(* IEC 61131-3 sources: ironplc-benchmarks/compat_out (part 34) *)

(*
version 1.1	15 sep 2007
programmer 	hugo
tested by		tobias

FT_TN7 is delay function, it will delay a signal by a specified time : T and will store 64 values of in before they are put thru to out.
if lower resolution is needed, pls use FT_TN8 or FT_TN16 instead.

*)
(* @END_DECLARATION := '0' *)
(* read system time *)
tx := DWORD_TO_TIME(T_PLC_MS());

trig := FALSE;
IF NOT init THEN
	x[cnt] := in;
	init := TRUE;
	last := tx;
ELSIF tx - last >= T / length THEN
	IF cnt = length - 1 THEN cnt := 0; ELSE cnt := cnt + 1; END_IF;
	Out := X[cnt];
	x[cnt] := in;
	last := tx;
	trig := TRUE;
END_IF;

(* revision history
hm		1. jan 2007		rev 1.0
	original version

hm		16. sep 2007	rev 1.1
	changes time() to T_plc_ms() for compatibility reasons

*)
END_FUNCTION_BLOCK

(* @NESTEDCOMMENTS := 'Yes' *)
(* @PATH := '\/Engineering\/control' *)
(* @OBJECTFLAGS := '0, 8' *)
(* @SYMFILEFLAGS := '2048' *)
FUNCTION_BLOCK FT_TN8
VAR_INPUT
	in : REAL;
	T : TIME;
END_VAR
VAR_OUTPUT
	out : REAL;
	trig: BOOL;
END_VAR
VAR
	length : INT := 8;
	X : ARRAY[0..7] OF REAL;
	cnt : INT;
	last : TIME;
	tx: TIME;
	init: BOOL;
END_VAR

(*
version 1.1	15 Sep 2007
programmer 	hugo
tested by		tobias

FT_TN8 is delay function, it will delay a signal by a specified time : T and will store 8 values of in before they are put thru to out.
if higher resolution is needed, pls use FT_TN16 or FT_TN64 instead.

*)
(* @END_DECLARATION := '0' *)
tx := DWORD_TO_TIME(T_PLC_MS());
trig := FALSE;
IF NOT init THEN
	x[cnt] := in;
	init := TRUE;
	last := tx;
ELSIF tx - last >= T / length THEN
	IF cnt = length - 1 THEN cnt := 0; ELSE cnt := cnt + 1; END_IF;
	Out := X[cnt];
	x[cnt] := in;
	last := tx;
	trig := TRUE;
END_IF;

(* revision history
hm		1. jan 2007		rev 1.0
	original version

hm		16. sep 2007	rev 1.1
	changes time() to T_plc_ms() for compatibility reasons

*)
END_FUNCTION_BLOCK

(* @NESTEDCOMMENTS := 'Yes' *)
(* @PATH := '\/Engineering\/control' *)
(* @OBJECTFLAGS := '0, 8' *)
(* @SYMFILEFLAGS := '2048' *)
FUNCTION_BLOCK HYST
VAR_INPUT
	In : REAL;
	ON : REAL;
	OFF : REAL;
END_VAR
VAR_OUTPUT
	Q : BOOL;
	win : BOOL;
END_VAR

(*
version 1.0	2. jun. 2008
programmer 	hugo
tested BY	oscat

This Hystereses function has two modes:
1. if on > off then Q will be switched high when in > on and switched low when in < off.
2. if on < off then Q will be switched high when in < on and switched low when in > off.
the output win will be high when in is between low and high.

*)
(* @END_DECLARATION := '0' *)
IF ON >= OFF THEN
	IF IN < OFF THEN
		Q := FALSE;
		WIN := FALSE;
	ELSIF  IN > ON THEN
		Q := TRUE;
		WIN := FALSE;
	ELSE
		WIN := TRUE;
	END_IF;
ELSE
	IF IN > OFF THEN
		Q := FALSE;
		WIN := FALSE;
	ELSIF  IN < ON THEN
		Q := TRUE;
		WIN := FALSE;
	ELSE
		WIN := TRUE;
	END_IF;
END_IF;

(* revision history
hm		2.  jun 2008	rev 1.0
	original version

*)
END_FUNCTION_BLOCK

(* @NESTEDCOMMENTS := 'Yes' *)
(* @PATH := '\/Engineering\/control' *)
(* @OBJECTFLAGS := '0, 8' *)
(* @SYMFILEFLAGS := '2048' *)
FUNCTION_BLOCK HYST_1
VAR_INPUT
	In : REAL;
	high : REAL;
	low : REAL;
END_VAR
VAR_OUTPUT
	Q : BOOL;
	win : BOOL;
END_VAR

(*
version 1.1	2. jun. 2008
programmer 	hugo
tested BY	oscat

this hysteresis function switches the output high if the input signal reaches obove high and will switch to low when the input falls back below low value.
a separate output mid is set if the input stays between low and high value.

*)
(* @END_DECLARATION := '0' *)
IF in < low THEN
	Q := FALSE;
	win := FALSE;
ELSIF in > high THEN
	Q := TRUE;
	win := FALSE;
ELSE
	win := TRUE;
END_IF;

(* revision history
hm		4.  aug. 2006	rev 1.0
	original version

hm		2. jun. 2008	rev 1.1
	improved performance
*)
END_FUNCTION_BLOCK

(* @NESTEDCOMMENTS := 'Yes' *)
(* @PATH := '\/Engineering\/control' *)
(* @OBJECTFLAGS := '0, 8' *)
(* @SYMFILEFLAGS := '2048' *)
FUNCTION_BLOCK HYST_2
VAR_INPUT
	IN : REAL;
	VAL : REAL;
	HYS : REAL;
END_VAR
VAR_OUTPUT
	Q : BOOL;
	WIN: BOOL;
END_VAR
VAR
	tmp: REAL;
END_VAR

(*
version 1.2	2. jun. 2008
programmer 	oscat
tested BY	oscat

this hysteresis function switches the output high if the input signal reaches obove val + hys/2 and will switch to low when the input falls back below val - hys/2 value.
a separate output mid is set if the input stays between low and high value.

*)
(* @END_DECLARATION := '0' *)
tmp := val - hys * 0.5;
IF in < tmp THEN
	Q := FALSE;
	win := FALSE;
ELSIF in > tmp + hys THEN
	Q := TRUE;
	win := FALSE;
ELSE
	win := TRUE;
END_IF;

(* revision history
hm		4. aug 2006	rev 1.0
	original version

hm		5. jan 2008	rev 1.1
	improved code for better performance

hm		2. jun. 2008	rev 1.2
	improved performance
*)
END_FUNCTION_BLOCK

(* @NESTEDCOMMENTS := 'Yes' *)
(* @PATH := '\/Engineering\/control' *)
(* @OBJECTFLAGS := '0, 8' *)
(* @SYMFILEFLAGS := '2048' *)
FUNCTION_BLOCK HYST_3
VAR_INPUT
	in : REAL;
	hyst : REAL;
	val1 : REAL;
	val2 : REAL;
END_VAR
VAR_OUTPUT
	Q1 : BOOL;
	Q2 : BOOL;
END_VAR
VAR
	X: REAL;
END_VAR

(*
version 1.2	5 jan 2008
programmer 	oscat
tested BY	oscat

this is a double hysteresis function. Out1 follows a hysteresis function defined by val1and hyst, while out 2 follows val2 and hyst.
if the input signal is between the two hysteresis switches (val1 and val2) then non of the outputs is active.

*)
(* @END_DECLARATION := '0' *)
X := hyst * 0.5;
IF in < val1 - X THEN
	q1 := TRUE;
ELSIF in > val1 + X THEN
	q1 := FALSE;
END_IF;
IF in < val2 - X THEN
	q2 := FALSE;
ELSIF in > val2 + X THEN
	q2 := TRUE;
END_IF;

(* revision history
hm	22. jan 2007	rev 1.0
	original version

hm	27. dec 2007	rev 1.1
	changed code for better performance

hm	5. jan 2008	rev 1.2
	further performance iprovements

*)

END_FUNCTION_BLOCK

(* @NESTEDCOMMENTS := 'Yes' *)
(* @PATH := '\/Engineering\/control' *)
(* @OBJECTFLAGS := '0, 8' *)
(* @SYMFILEFLAGS := '2048' *)
FUNCTION_BLOCK INTEGRATE
VAR_INPUT
	E : BOOL := TRUE;
	X : REAL;
	K : REAL := 1.0;
END_VAR
VAR_IN_OUT
	Y : REAL;
END_VAR
VAR
	X_last : REAL;
	init: BOOL;
	last: DWORD;
	tx: DWORD;
END_VAR

(*
version 1.0	3. nov. 2008
programmer 	hugo
tested by	oscat

integrate is a plain integrator with I/O for out.

*)
(* @END_DECLARATION := '0' *)
(*read system time *)
tx := T_PLC_MS();

IF NOT init THEN
	init := TRUE;
	X_last := X;
ELSIF E THEN
	Y := (X + X_LAST) * 0.5E-3 * DWORD_TO_REAL(tx-last) * K + Y;
	X_last := X;
END_IF;
last := tx;

(*
hm 3. nov. 2008	rev 1.0
original version

*)

END_FUNCTION_BLOCK

(* @NESTEDCOMMENTS := 'Yes' *)
(* @PATH := '\/Engineering\/conversion' *)
(* @OBJECTFLAGS := '0, 8' *)
(* @SYMFILEFLAGS := '2048' *)
FUNCTION_BLOCK ASTRO
VAR_INPUT
	m : REAL;
	AE : REAL;
	PC : REAL;
	LJ : REAL;
END_VAR
VAR_OUTPUT
	Ym : REAL;
	YAE : REAL;
	YPC : REAL;
	YLJ : REAL;
END_VAR

(*
version 1.1	11. mar. 2009
programmer 	hugo
tested by		oscat

this function converts different length units
any unused input can simply be left open.
different inputs connected at the same time will be added up.

*)
(* @END_DECLARATION := '0' *)
YAE :=	AE
		+ m * 6.6845871535E-012
		+ PC * 206265.0
		+ LJ * 63240.0;
Ym := YAE * 149.597870E9;
YPC := YAE * 4.8481322570E-006;
YLJ := YAE * 1.5812776724E-005;

(*
L�nge Meter m SI-Basiseinheit
Astronomische Einheit* AE 1 AE = 149,597 870 � E9 m
Parsec pc 1 pc = 206265 AE = 30,857 � E15 m
Lichtjahr Lj 1 Lj = 9,460 530 � E15 m = 63240 AE = 0,306 59 pc
�ngstr�m � 1 � = E�l0 m
typograph. Punkt p 1 p = 0,376 065 mm � im Druckereigewerbe
inch** in 1 in = 2,54 � E�2 m = 25,4 mm***
foot ft 1 ft = 0,3048 m = 30,48 cm
yard yd 1 yd = 0,9144 m
mile mile 1 mile = 1609,344 m
Internat. Seemeile sm 1 sm = 1852 m
Fathom fm 1 fm = 1,829 m � in der Seeschifffahrt
*)

(* revision history

hm	27. mar. 2007	rev 1.0
	original version

hm	11. mar. 2009	rev 1.1
	improved code

*)

END_FUNCTION_BLOCK

(* @NESTEDCOMMENTS := 'Yes' *)
(* @PATH := '\/Engineering\/conversion' *)
(* @OBJECTFLAGS := '0, 8' *)
(* @SYMFILEFLAGS := '2048' *)
FUNCTION BFT_TO_MS : REAL
VAR_INPUT
	BFT : INT;
END_VAR

(*
version 1.0	12. jun 2008
programmer 	hugo
tested by		oscdat

this function converts wind speed from beaufort to m/s
*)
(* @END_DECLARATION := '0' *)
BFT_TO_MS := EXPT(BFT, 1.5) * 0.836;

(* revision history
hm	12. 6. 2008		rev 1.0
	original version

*)
END_FUNCTION

(* @NESTEDCOMMENTS := 'Yes' *)
(* @PATH := '\/Engineering\/conversion' *)
(* @OBJECTFLAGS := '0, 8' *)
(* @SYMFILEFLAGS := '2048' *)
FUNCTION C_TO_F : REAL
VAR_INPUT
	celsius : REAL;
END_VAR

(*
version 1.1	11. mar. 2009
programmer 	hugo
tested by		tobias

this function converts celsius  to fahrenheit

*)
(* @END_DECLARATION := '0' *)
C_TO_F := celsius * 1.8 + 32.0;

(* revision history

hm	4. aug. 2006	rev 1.0
	original version

hm	11. mar. 2009	rev 1.1
	real constants updated to new systax using dot

*)
END_FUNCTION

(* @NESTEDCOMMENTS := 'Yes' *)
(* @PATH := '\/Engineering\/conversion' *)
(* @OBJECTFLAGS := '0, 8' *)
(* @SYMFILEFLAGS := '2048' *)
FUNCTION C_TO_K : REAL
VAR_INPUT
	Celsius : REAL;
END_VAR

(*
version 1.1	19. aug 2009
programmer 	hugo
tested by		tobias

this function converts celsius to kelvin
*)
(* @END_DECLARATION := '0' *)
C_TO_K := Celsius - phys.T0;

(* revision history

hm	4. aug 2006	rev 1.0
	original version

hm	19. aug 2009	rev 1.1
	fixed calculation error

*)

END_FUNCTION

(* @NESTEDCOMMENTS := 'Yes' *)
(* @PATH := '\/Engineering\/conversion' *)
(* @OBJECTFLAGS := '0, 8' *)
(* @SYMFILEFLAGS := '2048' *)
FUNCTION DEG_TO_DIR : STRING[3]
VAR_INPUT
	DEG : INT;
	N : INT;
	L : INT;
END_VAR
VAR
	ly: INT;
END_VAR

(*
version 1.1	22. oct. 2008
programmer 	hugo
tested by		oscat

this function converts degrees in compass direction.
the function supports output in english (L=0) and german (L=1).

*)
(* @END_DECLARATION := '0' *)
IF L = 0 THEN ly := LANGUAGE.DEFAULT; ELSE ly := MIN(L, LANGUAGE.LMAX); END_IF;
DEG_TO_DIR := LANGUAGE.DIRS[ly, ((SHL(DEG,N-1) + 45) / 90) MOD SHL(INT#2,N)*SHR(INT#8,N)];

(*
DIR := ((SHL(DEG,N-1) + 45) / 90) MOD SHL(INT#2,N);
explanation :
DIR is calculated BY the following formula:
DIR := ((DIR + 45) / 90) MOD 4 if N = 1 digit
North = 0, East = 1 ....
DIR := ((DIR + 22,5) / 45) MOD 8 if N = 2 digit
convert to integer calculation
DIR := ((DIR*2 + 45) / 90) MOD 8
N = 0, NE = 1 ....
ther above formula replaces 2^N with shift for performance
*)

(* revision histroy
hm	11. jun. 2008	rev 1.0
	original release

hm	22. oct. 2008	rev 1.1
	changed size of string variables to 30
*)
END_FUNCTION

(* @NESTEDCOMMENTS := 'Yes' *)
(* @PATH := '\/Engineering\/conversion' *)
(* @OBJECTFLAGS := '0, 8' *)
(* @SYMFILEFLAGS := '2048' *)
FUNCTION DIR_TO_DEG : INT
VAR_INPUT
	DIR : STRING[3];
	L : INT;
END_VAR
VAR
	ly: INT;
	i : INT;
END_VAR

(*
version 1.1	22. oct. 2008
programmer 	hugo
tested by	oscat

this function converts compass directions to degrees
it will recognize up to 3 letter directions in english and german writing.

*)
(* @END_DECLARATION := '0' *)
IF L = 0 THEN ly := LANGUAGE.DEFAULT; ELSE ly := MIN(L, LANGUAGE.LMAX); END_IF;
FOR i := 0 TO 15 DO
	IF language.DIRS[ly, i] = DIR THEN EXIT; END_IF;
END_FOR;
DIR_TO_DEG := SHR(i * 45 + 1, 1);

(* revision histroy
hm	22. oct. 2008	rev 1.1
	original release

*)
END_FUNCTION

(* @NESTEDCOMMENTS := 'Yes' *)
(* @PATH := '\/Engineering\/conversion' *)
(* @OBJECTFLAGS := '0, 8' *)
(* @SYMFILEFLAGS := '2048' *)
FUNCTION_BLOCK ENERGY
VAR_INPUT
	J : REAL;
	C : REAL;
	Wh : REAL;
END_VAR
VAR_OUTPUT
	YJ : REAL;
	YC : REAL;
	YWh : REAL;
END_VAR

(*
version 1.2	16. jan. 2010
programmer 	hugo
tested by		oscat

this function converts different energy units
any unused input can simply be left open.
different inputs connected at the same time will be added up.
*)
(* @END_DECLARATION := '0' *)
YJ := J + Wh * 3600.0 + C * 4.1868;
YC := YJ * 0.238845896627496;
YWh := YJ * 2.7777777778E-004;

(*
Arbeit, Energie, Joule* J 1 J = 1 N � m = 1 W � s = (1/3,6) E�6 kW � h = 1 kg � m2/s2
W�rmemenge Kilowattstunde kW � h 1 kW � h = 3,6 MJ = 860 kcal
Elektronvolt eV 1 eV = 160,218 92 E�21 J
Erg erg 1 erg = 1E�7 J
Kalorie calorie 1 calalorie = 4,1868 J = 1,163 E�3 W � h
Therm therm 1 therm = 105,50 � 106 J
*)

(* revision history

hm	27. mar. 2007	rev 1.0
	original version

hm	11. mar. 2009	rev 1.1
	improved code

hm 16. jan 2010	rev 1.2
	avoid the string cal in comments for codesys import bug

*)
END_FUNCTION_BLOCK

(* @NESTEDCOMMENTS := 'Yes' *)
(* @PATH := '\/Engineering\/conversion' *)
(* @OBJECTFLAGS := '0, 8' *)
(* @SYMFILEFLAGS := '2048' *)
FUNCTION F_TO_C : REAL
VAR_INPUT
	fahrenheit : REAL;
END_VAR

(*
version 1.1	11. mar. 2009
programmer 	hugo
tested BY		tobias

this FUNCTION converts fahrenheit TO celsius

*)
(* @END_DECLARATION := '0' *)
F_TO_C := (fahrenheit - 32.0) * 0.5555555555555;

(* revision history
hm	4. aug 2006	rev 1.0
	original version

hm	11. mar. 2009	rev 1.1
	real constants updated to new systax using dot

*)
END_FUNCTION

(* @NESTEDCOMMENTS := 'Yes' *)
(* @PATH := '\/Engineering\/conversion' *)
(* @OBJECTFLAGS := '0, 8' *)
(* @SYMFILEFLAGS := '2048' *)
FUNCTION F_TO_OM : REAL
VAR_INPUT
	F : REAL;
END_VAR

(*
version 1.1	18. oct. 2008
programmer 	hugo
tested by	oscat

this function converts frequency to Omega F
Omega = 2*PI*F
*)
(* @END_DECLARATION := '0' *)
F_TO_OM := math.PI2 * F;

(* revision history
hm	22. jan. 2007	rev 1.0
	original version

hm	18. oct. 2008	rev 1.1
	unsing math constants

*)
END_FUNCTION

(* @NESTEDCOMMENTS := 'Yes' *)
(* @PATH := '\/Engineering\/conversion' *)
(* @OBJECTFLAGS := '0, 8' *)
(* @SYMFILEFLAGS := '2048' *)
FUNCTION F_TO_PT : TIME
VAR_INPUT
	F : REAL;
END_VAR

(*
version 1.1	11. mar. 2009
programmer 	hugo
tested by		tobias

this function converts frequency to periode time
*)
(* @END_DECLARATION := '0' *)
F_TO_PT := DWORD_TO_TIME(REAL_TO_DWORD(1.0 / F * 1000.0));

(* revision history

hm	4. aug. 2006	rev 1.0
	original version

hm	11. mar. 2009	rev 1.1
	real constants updated to new systax using dot

*)

END_FUNCTION

(* @NESTEDCOMMENTS := 'Yes' *)
(* @PATH := '\/Engineering\/conversion' *)
(* @OBJECTFLAGS := '0, 8' *)
(* @SYMFILEFLAGS := '2048' *)
FUNCTION GEO_TO_DEG : REAL
VAR_INPUT
	D : INT;
	M : INT;
	SEC : REAL;
END_VAR

(*
version 1.0	22. jan. 2009
programmer 	hugo
tested by		oscat

this function converts degrees, minutes seconds to decimal degrees.

*)
(* @END_DECLARATION := '0' *)
GEO_TO_DEG := INT_TO_REAL(D) + INT_TO_REAL(M) * 0.016666666666667 + sec * 0.00027777777777778;

(* revision histroy
hm	22. jan. 2009	rev 1.0
	original release

*)
END_FUNCTION

(* @NESTEDCOMMENTS := 'Yes' *)
(* @PATH := '\/Engineering\/conversion' *)
(* @OBJECTFLAGS := '0, 8' *)
(* @SYMFILEFLAGS := '2048' *)
FUNCTION K_TO_C : REAL
VAR_INPUT
	Kelvin : REAL;
END_VAR

(*
version 1.1	19. aug 2009
programmer 	hugo
tested by		tobias

this function converts kelvin to celsius

*)
(* @END_DECLARATION := '0' *)
K_TO_C := Kelvin + phys.T0;

(* revision history

hm	4. aug 2006	rev 1.0
	original version

hm	19. aug 2009	rev 1.1
	fixed calculation error

*)

END_FUNCTION

(* @NESTEDCOMMENTS := 'Yes' *)
(* @PATH := '\/Engineering\/conversion' *)
(* @OBJECTFLAGS := '0, 8' *)
(* @SYMFILEFLAGS := '2048' *)
FUNCTION KMH_TO_MS : REAL
VAR_INPUT
	kmh : REAL;
END_VAR

(*
version 1.1	6 jan 2007
programmer 	hugo
tested by		tobias

this function converts velocities from Kilometers / hour to Meters / Second

*)
(* @END_DECLARATION := '0' *)
KMH_TO_MS := kmh * 0.2777777777777;

(* revision history
hm	4. feb 2007		rev 1.0
	original version

hm	6. jan 2008		rev 1.1
	improved performance

*)

END_FUNCTION

(* @NESTEDCOMMENTS := 'Yes' *)
(* @PATH := '\/Engineering\/conversion' *)
(* @OBJECTFLAGS := '0, 8' *)
(* @SYMFILEFLAGS := '2048' *)
FUNCTION_BLOCK LENGTH
VAR_INPUT
	m : REAL;
	p : REAL;
	in : REAL;
	ft : REAL;
	yd : REAL;
	mile : REAL;
	sm : REAL;
	fm : REAL;
END_VAR
VAR_OUTPUT
	Ym : REAL;
	Yp : REAL;
	Yin : REAL;
	Yft : REAL;
	Yyd : REAL;
	Ymile : REAL;
	Ysm : REAL;
	Yfm : REAL;
END_VAR

(*
version 1.1	11. mar. 2009
programmer 	hugo
tested by		oscat

this function converts different length units
any unused input can simply be left open.
different inputs connected at the same time will be added up.

*)
(* @END_DECLARATION := '0' *)
Ym :=	m
		+ p * 0.000376065
		+ in * 0.0254
		+ ft * 0.3048
		+ yd * 0.9144
		+ mile * 1609.344
		+ sm * 1852.0
		+ fm * 1.829;
Yp := Ym * 2659.11478068951;
Yin := Ym * 39.37007874016;
Yft := Ym * 3.28083989501;
Yyd := Ym * 1.09361329834;
Ymile := Ym * 0.00062137119;
Ysm := Ym * 0.00053995680;
Yfm := Ym * 0.54674685621;

(*
L�nge Meter m SI-Basiseinheit
Astronomische Einheit* AE 1 AE = 149,597 870 � E9 m
Parsec pc 1 pc = 206265 AE = 30,857 � E15 m
Lichtjahr Lj 1 Lj = 9,460 530 � E15 m = 63240 AE = 0,306 59 pc
�ngstr�m � 1 � = E�l0 m
typograph. Punkt p 1 p = 0,376 065 mm � im Druckereigewerbe
inch** in 1 in = 2,54 � E�2 m = 25,4 mm***
foot ft 1 ft = 0,3048 m = 30,48 cm
yard yd 1 yd = 0,9144 m
mile mile 1 mile = 1609,344 m
Internat. Seemeile sm 1 sm = 1852 m
Fathom fm 1 fm = 1,829 m � in der Seeschifffahrt
*)

(* revision history

hm	27. mar. 2007	rev 1.0
	original version

hm	11. mar. 2009	rev 1.1
	improved code

*)

END_FUNCTION_BLOCK

(* @NESTEDCOMMENTS := 'Yes' *)
(* @PATH := '\/Engineering\/conversion' *)
(* @OBJECTFLAGS := '0, 8' *)
(* @SYMFILEFLAGS := '2048' *)
FUNCTION MS_TO_BFT : INT
VAR_INPUT
	MS : REAL;
END_VAR

(*
version 1.0	12. jun 2008
programmer 	hugo
tested by	oscdat

this function converts wind speed from M/s to beaufort
*)
(* @END_DECLARATION := '0' *)
MS_TO_BFT := REAL_TO_INT(EXPT(MS * 1.196172, 0.666667));

(* revision history
hm	12. 6. 2008		rev 1.0
	original version

*)
END_FUNCTION

(* @NESTEDCOMMENTS := 'Yes' *)
(* @PATH := '\/Engineering\/conversion' *)
(* @OBJECTFLAGS := '0, 8' *)
(* @SYMFILEFLAGS := '2048' *)
FUNCTION MS_TO_KMH : REAL
VAR_INPUT
	ms : REAL;
END_VAR

(*
version 1.0	4 Feb 2007
programmer 	hugo
tested by		tobias

this function converts velocities from Meters / Second to Kilometers / hour.

*)
(* @END_DECLARATION := '0' *)
MS_TO_KMH := ms * 3.6;

END_FUNCTION

(* @NESTEDCOMMENTS := 'Yes' *)
(* @PATH := '\/Engineering\/conversion' *)
(* @OBJECTFLAGS := '0, 8' *)
(* @SYMFILEFLAGS := '2048' *)
FUNCTION OM_TO_F : REAL
VAR_INPUT
	OM : REAL;
END_VAR

(*
version 1.1	18. oct. 2008
programmer 	hugo
tested by		tobias

this function converts Omega F to frequency
F = OM / (2*PI)
*)
(* @END_DECLARATION := '0' *)
OM_TO_F := OM / math.PI2;

(* revision history
hm	22. jan. 2007	rev 1.0
	original version

hm	18. oct. 2008	rev 1.1
	using math constants

*)
END_FUNCTION

(* @NESTEDCOMMENTS := 'Yes' *)
(* @PATH := '\/Engineering\/conversion' *)
(* @OBJECTFLAGS := '0, 8' *)
(* @SYMFILEFLAGS := '2048' *)
FUNCTION_BLOCK PRESSURE
VAR_INPUT
	mws : REAL;
	torr : REAL;
	att : REAL;
	atm : REAL;
	pa : REAL;
	bar : REAL;
END_VAR
VAR_OUTPUT
	Ymws : REAL;
	Ytorr : REAL;
	Yatt : REAL;
	Yatm : REAL;
	Ypa : REAL;
	Ybar : REAL;
END_VAR

(*
version 1.1	11. mar. 2009
programmer 	hugo
tested by		oscat

this function converts different pressure units
any unused input can simply be left open.
different inputs connected at the same time will be added up.
*)
(* @END_DECLARATION := '0' *)
Ybar := bar +
		pa * 1.0E-5 +
		0.980665 * att +
		1.01325 * atm +
		0.001333224 * torr +
		0.0980665 * mws;
Ymws := ybar * 10.1971621297793;
Ytorr := ybar * 750.0615050434140;
Yatt := ybar * 1.0197162129779;
yatm := ybar * 0.9869232667160;
Ypa := ybar * 100000.0;

(*
Druck, Pascal Pa 1 Pa = 1 N/m2 = 1 kg/(s2 �E m) . 0,75 �E 10.2 mmHg
mechanische 1 MPa = 1 N/mm2 . fur Festigkeitsangaben
Spannung Bar bar 1 bar = 105 Pa = 103 mbar = 105 kg/(s2 �E m)
Millimeter- mmHg 1 mmHg = 133,322 Pa = 1,333 22 mbar
Quecksilbersaule . nur in Heilkunde zulassig
physik. Atmosphare atm 1 atm = 1,013 25 bar
techn. Atmosphare at 1 at = 1 kp/cm2 = 0,980665 bar
Torr Torr 1 Torr = (101325/760) Pa = 1,333224 mbar
Meter-Wassersaule mWS 1 mWS = 9806,65 Pa = 98,0665 mbar
psi lbf/in2 1 lbf/in2 = 68,947 57 mbar = 6894,757 Pa

*)

(* revision history

hm	27. mar. 2007	rev 1.0
	original version

hm	11. mar. 2009	rev 1.1
	improved code

*)
END_FUNCTION_BLOCK

(* @NESTEDCOMMENTS := 'Yes' *)
(* @PATH := '\/Engineering\/conversion' *)
(* @OBJECTFLAGS := '0, 8' *)
(* @SYMFILEFLAGS := '2048' *)
FUNCTION PT_TO_F : REAL
VAR_INPUT
	PT : TIME;
END_VAR

(*
version 1.1	11. mar. 2009
programmer 	hugo
tested by		tobias

this function converts periode time to frequency
*)
(* @END_DECLARATION := '0' *)
PT_TO_F := 1000.0 / DWORD_TO_REAL(TIME_TO_DWORD(PT));

(*	revision history
hm	4. aug. 2006	rev 1.0
	original version

hm	11. mar. 2009	rev 1.1
	real constants updated to new systax using dot

*)

END_FUNCTION

(* @NESTEDCOMMENTS := 'Yes' *)
(* @PATH := '\/Engineering\/conversion' *)
(* @OBJECTFLAGS := '0, 8' *)
(* @SYMFILEFLAGS := '2048' *)
FUNCTION_BLOCK SPEED
VAR_INPUT
	ms : REAL;
	kmh : REAL;
	kn : REAL;
	mh : REAL;
END_VAR
VAR_OUTPUT
	Yms : REAL;
	Ykmh : REAL;
	Ykn : REAL;
	Ymh : REAL;
END_VAR

(*
version 1.1	11. mar. 2009
programmer 	hugo
tested by		oscat

this function converts different speed units
any unused input can simply be left open.
different inputs connected at the same time will be added up.

*)
(* @END_DECLARATION := '0' *)
Yms := ms +
		kmh * 0.27777777777778 +
		kn * 0.5144444 +
		mh * 0.44704;
Ykmh := Yms * 3.6;
Ykn := Yms * 1.94384466037535;
Ymh := Yms * 2.23693629205440;

(*
Geschwindigkeit Meter durch Sekunde m/s 1 m/s = 3,6 km/h
km durch (pro) Stunde, nicht �Stundenkilometer� verwenden
Knoten kn 1 kn = 1 sm/h = 0,5144 m/s

*)

(* revision history
hm	27. mar. 2009	rev 1.0
	original version

hm	11. mar. 2009	rev 1.1
	improved code

*)
END_FUNCTION_BLOCK

(* @NESTEDCOMMENTS := 'Yes' *)
(* @PATH := '\/Engineering\/conversion' *)
(* @OBJECTFLAGS := '0, 8' *)
(* @SYMFILEFLAGS := '2048' *)
FUNCTION_BLOCK TEMPERATURE
VAR_INPUT
	K : REAL;
	C : REAL := -273.15;
	F : REAL := -459.67;
	Re : REAL := -218.52;
	Ra : REAL;
END_VAR
VAR_OUTPUT
	YK : REAL;
	YC : REAL;
	YF : REAL;
	YRe : REAL;
	YRa : REAL;
END_VAR

(*
version 1.0	21 feb 2008
programmer 	hugo
tested by	oscat

this function converts different temperature units
any unused input can simply be left open.
different inputs connected at the same time will be added up.

*)
(* @END_DECLARATION := '0' *)
YK := K + (C + 273.15) + (F + 459.67) * 0.555555555555 + (Re * 1.25 + 273.15) + (Ra * 0.555555555555);
YC := YK -273.15;
YF := YK * 1.8 - 459.67;
YRe := (YK - 273.15) * 0.8;
YRa := YK * 1.8;

(* revision history
hm	21. feb. 2008	rev 1.0
	original version

*)
END_FUNCTION_BLOCK

(* @NESTEDCOMMENTS := 'Yes' *)
(* @PATH := '\/Engineering\/measurements' *)
(* @OBJECTFLAGS := '0, 8' *)
(* @SYMFILEFLAGS := '2048' *)
FUNCTION_BLOCK ALARM_2
VAR_INPUT
	X : REAL;
	LO_1 : REAL;
	HI_1 : REAL;
	LO_2 : REAL;
	HI_2 : REAL;
	HYS : REAL;
END_VAR
VAR_OUTPUT
	Q1_LO : BOOL;
	Q1_HI : BOOL;
	Q2_LO : BOOL;
	Q2_HI : BOOL;
END_VAR
VAR
	tmp: REAL;
END_VAR

(*
	version 1.1	11. mar. 2009
	programmer 	hugo
	tested BY		tobias

ALARM_2 will check two pairs of limits and signal when the input is above or below a set limit.
with the input HYS a hysteresis can be defined for all limits.

*)
(* @END_DECLARATION := '0' *)
tmp := X - Hys * 0.5;
IF tmp > LO_1 THEN Q1_LO := FALSE; END_IF;
IF tmp > LO_2 THEN Q2_LO := FALSE; END_IF;
IF tmp > HI_1 THEN Q1_HI := TRUE; END_IF;
IF tmp > HI_2 THEN Q2_HI := TRUE; END_IF;
tmp := tmp + hys;
IF tmp < LO_1 THEN Q1_LO := TRUE; END_IF;
IF tmp < LO_2 THEN Q2_LO := TRUE; END_IF;
IF tmp < HI_1 THEN Q1_HI := FALSE; END_IF;
IF tmp < HI_2 THEN Q2_HI := FALSE; END_IF;

(* revision history
hm	19. may. 2008		rev 1.0
	original version

hm	11. mar. 2009	rev 1.1
	improved code
*)

END_FUNCTION_BLOCK

(* @NESTEDCOMMENTS := 'Yes' *)
(* @PATH := '\/Engineering\/measurements' *)
(* @OBJECTFLAGS := '0, 8' *)
(* @SYMFILEFLAGS := '2048' *)
FUNCTION_BLOCK BAR_GRAPH
VAR_INPUT
	X : REAL;
	rst : BOOL;
END_VAR
VAR_INPUT (* CONSTANT *)
	trigger_Low : REAL;
	trigger_High : REAL;
	Alarm_low : BOOL;
	Alarm_high : BOOL;
	log_scale : BOOL;
END_VAR
VAR_OUTPUT
	LOW, Q1, Q2, Q3, Q4, Q5, Q6, HIGH : BOOL;
	Alarm : BOOL;
	Status : BYTE;
END_VAR
VAR
	init : BOOL;
	T1, T2, T3, T4, T5 : REAL;
END_VAR
VAR_TEMP
	temp : REAL;
END_VAR

(*
	version 1.2	6 jan 2008
	programmer 	hugo
	tested BY	hans

bar graph is a muti window comparator which displays an analog input signal on 8 digital outputs.
only one output is active a any given time depending on the value of the input signal.
the output can be of linear or logarithmic scale.

*)
(* @END_DECLARATION := '0' *)
IF NOT init THEN
	init := TRUE;
	IF log_scale THEN
		temp := EXP(LN(Trigger_high / Trigger_low) * 0.166666666666666666666);
		T1 := trigger_low * temp;
		T2 := T1 * temp;
		T3 := T2 * temp;
		T4 := T3 * temp;
		T5 := T4 * temp;
	ELSE
		temp := (trigger_high - trigger_low) * 0.142857142;
		T1 := trigger_low + temp;
		T2 := T1 + temp;
		T3 := T2 + temp;
		T4 := T3 + temp;
		T5 := T4 + temp;
	END_IF;
END_IF;

(* clear outputs before checking *)
Q1 := FALSE;
Q2 := FALSE;
Q3 := FALSE;
Q4 := FALSE;
Q5 := FALSE;
Q6 := FALSE;
status := 110;

(* low, high and alarm can only be cleared with rst depending on alarm_low and alarm_high *)
IF NOT alarm_low THEN low := FALSE; END_IF;
IF NOT alarm_high THEN high := FALSE; END_IF;
IF rst THEN
	alarm := FALSE;
	low := FALSE;
	high := FALSE;
END_IF;

(* check and set outputs *)
IF X < trigger_low THEN
	Low := TRUE;
	status := 111;
	IF alarm_low THEN
		alarm := TRUE;
		status := 1;
	END_IF;
ELSIF X < T1 THEN
	Q1 := TRUE;
ELSIF x < t2 THEN
	Q2 := TRUE;
ELSIF x < t3 THEN
	Q3 := TRUE;
ELSIF x < T4 THEN
	Q4 := TRUE;
ELSIF x < T5 THEN
	q5 := TRUE;
ELSIF x < trigger_high THEN
	q6 := TRUE;
ELSE
	high := TRUE;
	status := 112;
	IF alarm_high THEN
		alarm := TRUE;
		status := 2;
	END_IF;
END_IF;

(* revision history
hm	22. feb 2007	rev 1.0
	original version

hm	2. dec 2007		rev 1.1
	chaged code for better performance

hm	6. jan 2008		rev 1.2
	further performance improvement

*)
END_FUNCTION_BLOCK

(* @NESTEDCOMMENTS := 'Yes' *)
(* @PATH := '\/Engineering\/measurements' *)
(* @OBJECTFLAGS := '0, 8' *)
(* @SYMFILEFLAGS := '2048' *)
FUNCTION_BLOCK CALIBRATE
VAR_INPUT
	X : REAL;
	CO : BOOL;
	CS : BOOL;
END_VAR
VAR_INPUT (* CONSTANT *)
	Y_Offset : REAL;
	Y_Scale : REAL;
END_VAR
VAR_OUTPUT
	Y : REAL;
END_VAR
VAR RETAIN
	offset : REAL;
	Scale : REAL := 1.0;
END_VAR

(*
	version 1.3	11. mar. 2009
	programmer 	hugo
	tested BY		hans

Calibrate allows for offset and scale calibration of an analog input.
offset is calibrated to a stored reference Y_offset while CO is true.
after the offset is calibrated, scale can be calibrated to a reference value Y_scale while CS is true.
*)
(* @END_DECLARATION := '0' *)
(* check for calibration *)
IF CO THEN
	OFFSET := Y_Offset - X;
ELSIF CS THEN
	SCALE := Y_scale / (X + OFFSET);
END_IF;
(* calculate output *)
Y := (X + OFFSET) * SCALE;

(* revision history
hm 22.2.2007		rev 1.2
	changed VAR RETAIN PERSISTENT to VAR RETAIN for better compatibility
	wago lon contollers do not support persisitent

hm	11. mar. 2009	rev 1.3
	changed real constants to use dot syntax

*)
END_FUNCTION_BLOCK

(* @NESTEDCOMMENTS := 'Yes' *)
(* @PATH := '\/Engineering\/measurements' *)
(* @OBJECTFLAGS := '0, 8' *)
(* @SYMFILEFLAGS := '2048' *)
FUNCTION_BLOCK CYCLE_TIME
VAR_INPUT
	RST : BOOL;
END_VAR
VAR_OUTPUT
	ct_min : TIME;
	ct_max : TIME;
	ct_last : TIME;
	systime : TIME;
	sysdays : INT;
	cycles : DWORD;
END_VAR
VAR
	last_cycle : TIME;
	tx: TIME;
	init: BOOL;
END_VAR

(*
	version 1.2	16 sep 2007
	programmer 	hugo
	tested BY		hans

this function block measures the cycle time and displays the last, min and max cycle time of the current task.
the resolution is 1ms.
the cycles output is a dword counter which counts the cycles.
a rst pulse on the input will reset all data.

*)
(* @END_DECLARATION := '0' *)
tx := DWORD_TO_TIME(T_PLC_MS()) - last_cycle;
IF rst THEN
	ct_min := t#10h;
	ct_max := t#0ms;
	cycles := 0;
ELSIF last_cycle > t#0s THEN
	IF tx < ct_min THEN ct_min := tx;
	ELSIF tx > ct_max THEN ct_max := tx;
	END_IF;
	ct_last := tx;
ELSIF ct_min = t#0s THEN
	ct_min := t#0s - t#1ms;
END_IF;
IF init THEN
	systime := systime + tx;
		IF systime >= t#1d THEN
			systime := systime - t#1d;
			sysdays := sysdays + 1;
		END_IF;
END_IF;
init := TRUE;
last_cycle := last_cycle + tx;
cycles := cycles + 1;

(*	revision history
hm 12.12.2006		rev 1.1
	added cycles output, a dword cycle counter.
hm 10.3.2007			rev 1.2
	changed initialization of ct_min to t#10h for compatibility with siemens s7

hm	16.9.2007		rev 1.2
	changed Time() in T_PLC_MS() for compatibility resons

*)
END_FUNCTION_BLOCK

(* @NESTEDCOMMENTS := 'Yes' *)
(* @PATH := '\/Engineering\/measurements' *)
(* @OBJECTFLAGS := '0, 8' *)
(* @SYMFILEFLAGS := '2048' *)
FUNCTION_BLOCK DT_SIMU
VAR_INPUT
	START : DT;
	SPEED : REAL := 1.0;
END_VAR
VAR_OUTPUT
	DTS : DT;
END_VAR
VAR
	tc : DWORD;
	init: BOOL;
	last: DWORD;
	tx: DWORD;
	td: DWORD;
END_VAR

(*
version 1.2	8. mar. 2009
programmer 	hugo
tested by		oscat

DT_SIMU simulates a real time clock and can be adjusted to different speeds
it can also be used in simulation to simulate a real time clock.
the peed of the clock can be increased or decreased to debug timers.
with the input start a start date-time can be specified.

*)
(* @END_DECLARATION := '0' *)
(* read system timer *)
tx := T_PLC_MS();
tc := REAL_TO_DWORD(DWORD_TO_REAL(tx - last) * speed);

IF NOT init THEN
	init := TRUE;
	DTS := Start;
	tc := 0;
	last := tx;
ELSIF SPEED = 0.0 THEN
	DTS := DWORD_TO_DT(DT_TO_DWORD(DTS) + 1);
ELSIF tc >= 1000 THEN
	td := (tc / 1000) * 1000;
	DTS := DTS + DWORD_TO_TIME(td);
	last := last + REAL_TO_DWORD(DWORD_TO_REAL(td) / speed);
END_IF;

(* revision history
hm	11. sep. 2008	rev 1.0
	original version

hm	16. nov	2008	rev 1.1
	added type conversions for compatibility reasons

hm	8.	mar. 2009	rev 1.2
	added increment by cycle mode

*)

END_FUNCTION_BLOCK

(* @NESTEDCOMMENTS := 'Yes' *)
(* @PATH := '\/Engineering\/measurements' *)
(* @OBJECTFLAGS := '0, 8' *)
(* @SYMFILEFLAGS := '2048' *)
FUNCTION_BLOCK FLOW_METER
VAR_INPUT
	VX : REAL;
	E : BOOL;
	RST : BOOL;
END_VAR
VAR_INPUT (* CONSTANT *)
	PULSE_MODE : BOOL;
	UPDATE_TIME : TIME := t#1s;
END_VAR
VAR_OUTPUT
	F : REAL;
END_VAR
VAR_IN_OUT
	X : REAL;
	Y : UDINT;
END_VAR
VAR
	tx, tl : TIME;
	int1 : INTEGRATE;
	init: BOOL;
	e_last : BOOL;
	tmp: INT;
	x_last : REAL;
	y_last : UDINT;
END_VAR

(*
version 1.0	23. jan. 2011
programmer 	hugo
tested by	oscat

Flow meter measures flow according to gated time or pulses.

*)

(* @END_DECLARATION := '0' *)
IF NOT init THEN	(* init on power up *)
	init := TRUE;
	tl := tx;
	x_last := X;
	y_last := Y;
	int1.K := 2.7777777777777777E-4;
END_IF;

(* run integrator *)
int1(E := NOT (RST OR PULSE_MODE) AND E, X := VX, Y := X);	(* gated operation *)

IF RST THEN		(* reset *)
	X := 0.0;
	Y := 0;
	tl := tx;
	x_last := 0.0;
	y_last := 0;
ELSIF E AND PULSE_MODE THEN	(* check for pulse mode *)
	IF NOT e_last THEN X := X + VX; END_IF;
END_IF;
e_last := E;

(* reduce X to be less than 1 and increase Y respectively *)
IF X > 1.0 THEN
	tmp := FLOOR(X);
	Y := Y + INT_TO_UDINT(tmp);
	X := X - INT_TO_REAL(tmp);
END_IF;

(* calculate the current flow *)
tx := DWORD_TO_TIME(T_PLC_MS());
IF tx - tl >= UPDATE_TIME AND UPDATE_TIME > t#0s THEN
	F := (UDINT_TO_REAL(Y - y_last) + X - x_last) / TIME_TO_REAL(tx - tl) * 3.6E6;
	y_last := Y;
	x_last := X;
	tl := tx;
END_IF;

(* revision history
hm	23. jan. 2011	rev 1.0
	original version

*)

END_FUNCTION_BLOCK

(* @NESTEDCOMMENTS := 'Yes' *)
(* @PATH := '\/Engineering\/measurements' *)
(* @OBJECTFLAGS := '0, 8' *)
(* @SYMFILEFLAGS := '2048' *)
FUNCTION_BLOCK M_D
VAR_INPUT
	start : BOOL;
	stop : BOOL;
	tmax : TIME := t#10d;
	rst: BOOL;
END_VAR
VAR_OUTPUT
	PT : TIME;
	ET : TIME;
	run : BOOL;
END_VAR
VAR
	edge : BOOL;
	T0 : TIME;
	tx: TIME;
	startup: BOOL;
END_VAR

(*
	version 1.2	27. feb. 2009
	programmer 	hugo
	tested BY	oscat

m_d measures the time between a rising edge on start to a rising edge on stop and returs the last measured value on the output PT.
a second output ET is starting from 0 at the rising edge of start and is counting up until the rising edge of stop occurs.
the asynchronous input rst can reset the outputs at any time.
tmax defines a timeout wich is the maximum measurable time between start and stop, if this time is exceeded the outputs will stay at 0.
*)
(* @END_DECLARATION := '0' *)
(* check for rst input *)
IF rst OR et >= tmax THEN
	pt := t#0ms;
	et := t#0ms;
	startup := FALSE;
	run := FALSE;
END_IF;

(* avoid timers to start when input is true at startup *)
IF NOT startup THEN
	edge := start;
	startup := TRUE;
END_IF;

(* read system timer *)
tx := DWORD_TO_TIME(T_PLC_MS());

(* detect rising edge on start *)
IF start AND NOT edge AND NOT stop THEN
	t0 := tx;
	run := TRUE;
	pt := t#0s;
ELSIF stop AND run THEN
	pt := et;
	run := FALSE;
END_IF;
edge := start;
IF run THEN et := tx - t0; END_IF;

(* revision history
hm		2.5.2007	rev 1.0
	original version

hm		16.9.2007	rev 1.1
	changes time() to T_plc_ms() for compatibility reasons

hm	27. feb 2009	rev 1.2
	deleted unnecessary init with 0
*)

END_FUNCTION_BLOCK

(* @NESTEDCOMMENTS := 'Yes' *)
(* @PATH := '\/Engineering\/measurements' *)
(* @OBJECTFLAGS := '0, 8' *)
(* @SYMFILEFLAGS := '2048' *)
FUNCTION_BLOCK M_T
VAR_INPUT
	IN : BOOL;
	TMAX : TIME := t#10d;
	RST : BOOL;
END_VAR
VAR_OUTPUT
	PT : TIME;
	ET: TIME;
END_VAR
VAR
	edge : BOOL;
	start : TIME;
	tx: TIME;
END_VAR

(*
version 1.4	10. mar. 2009
programmer 	hugo
tested BY		oscat

m_t measures the with of a high pulse and returs the last measured pulse width on output PT.
a second output ET is starting from 0 at the rising edge and counting up until the falling edge occurs and resetts et to 0.
the asynchrtonous input rst can reset the outputs at any time.
tmax defines a maximum measurable time, if this value is exceeded the outputs will be reset to 0.

*)
(* @END_DECLARATION := '0' *)
(* read system time *)
tx := DWORD_TO_TIME(T_PLC_MS());

IF RST OR ET >= TMAX THEN
	PT :=  t#0s;
	ET := t#0s;
ELSIF IN THEN
	IF NOT edge THEN start := tx; END_IF;
	ET := tx - start;
ELSE
	PT := ET;
END_IF;
edge := IN;

(* revision history
hm	4. aug. 2006	rev 1.0
	original version

hm	2. may. 2007	rev 1.1
	added init variable to avoid unreasonable measurement if falling edge occurs first.
	added et (elapsed time) output to count from 0 at rising edge until a falling edge resets et to 0.
	added reset input.

hm	16. sep. 2007	rev 1.2
	changes time() to T_plc_ms() for compatibility reasons

hm	17. dec. 2008	rev 1.3
	code optimized

hm	10. mar. 2009	rev 1.4
	removed nested comments
	removed double assignments

*)
END_FUNCTION_BLOCK

(* @NESTEDCOMMENTS := 'Yes' *)
(* @PATH := '\/Engineering\/measurements' *)
(* @OBJECTFLAGS := '0, 8' *)
(* @SYMFILEFLAGS := '2048' *)
FUNCTION_BLOCK M_TX
VAR_INPUT
	in: BOOL;
	tmax : TIME := t#10d;
	rst : BOOL;
END_VAR
VAR_OUTPUT
	TH : TIME;
	TL : TIME;
	DC : REAL;
	F: REAL;
	ET : TIME;
END_VAR
VAR
	edge : BOOL;
	start: TIME;
	stop:TIME;
	tx: TIME;
	rise : BOOL;
	fall : BOOL;
	startup: BOOL;
END_VAR

(*
	version 1.4	11. mar. 2009
	programmer 	oscat
	tested BY		oscat

this measures the timing of a signal
TH is the high pulse width
TL is the low pulse width
DC is the duty cycle
F is the frequency
ET will start at 0 with a rising edge and count up till the next rising edge starts from 0 again.
the acuracy depends on the cycle time of the sps and is limited to 1ms resolution.
an asynchronous reset can reset all outputs to 0 at any time.
the input tmax can configure a timeout for ET where the function block will outomatically reset itself.
tmx is predefined to 10 days.
*)
(* @END_DECLARATION := '0' *)
(* check FOR rst input *)
IF rst OR (et >= tmax) THEN
	rise := FALSE;
	fall := FALSE;
	startup := FALSE;
	th := t#0ms;
	tl := t#0ms;
	DC := 0.0;
	F := 0.0;
	ET := t#0s;
END_IF;

(* avoid timers to start when input is true at startup *)
IF NOT startup THEN
	edge := in;
	startup := TRUE;
END_IF;

(* read system timer *)
tx := DWORD_TO_TIME(T_PLC_MS());

(* edge trigger rising and falling edge *)
IF in XOR edge THEN
	edge := in;
	(* rising edge starts measurement *)
	IF in THEN
		start := Tx;
		rise := TRUE;
		IF fall THEN tl := start - stop; END_IF;
		IF th > t#0ms AND tl > t#0ms THEN
			dc := TIME_TO_REAL(th) / TIME_TO_REAL(th+tl);
			f := 1000.0 / TIME_TO_REAL(th + tl);
		END_IF;
	(* falling edge starts second cycle measurement *)
	ELSE
		stop := Tx;
		fall := TRUE;
		IF rise THEN th := stop - start; END_IF;
		IF th > t#0ms AND tl > t#0ms THEN
			dc := TIME_TO_REAL(th) /  TIME_TO_REAL(th+tl);
			f := 1000.0 / TIME_TO_REAL(th + tl);
		END_IF;
	END_IF;
END_IF;
IF rise THEN et := tx - start; END_IF;

(* revision history
hm	4. aug. 2006	rev 1.0
	original version

hm	2. mai. 2007	rev 1.1
	made sure that no undefined values would be measured at startup conditions
	added output et
	added rst input
	added tmax input

hm	16. sep. 2007	rev 1.2
	changes time() to T_plc_ms() for compatibility reasons

hm	27. feb. 2009	rev 1.3
	deleted unnecessary init with 0

hm	11. mar. 2009	rev 1.4
	changed real constants to use dot syntax

*)
END_FUNCTION_BLOCK

(* @NESTEDCOMMENTS := 'Yes' *)
(* @PATH := '\/Engineering\/measurements' *)
(* @OBJECTFLAGS := '0, 8' *)
(* @SYMFILEFLAGS := '2048' *)
FUNCTION_BLOCK METER
VAR_INPUT
	M1, M2 : REAL;
	I1, I2 : BOOL;
	D : REAL := 1.0;
	RST : BOOL;
END_VAR
VAR_IN_OUT
	MX : REAL;
END_VAR
VAR
	MR : REAL2;
	MX1, MX2 : REAL; (* current consumption value on M1 and M2 *)
	tx: DWORD;
	last: DWORD;
	tc: REAL;
	init: BOOL;
END_VAR

(*
	version 1.4	8. mar. 2009
	programmer 	oscat
	tested BY	oscat

METER measures usage of power or similar values the output MX is the sum of the inputs over time.
MX := sum over time of (I1 * P1 + I2 * P2)/D.
a simple example is the consumption counter for a 2 stage oil burner where stage 1 is 10KW and stage 2 is 20KW.
I1 and I2 decide which value is accounted for, I1 = True only counts P1, I2 is True counts P2
and I1 and I2 is true counts P1 and P2.
the meter can be used for all kind of consumption meters. P1 and P2 can change on the fly.

*)
(* @END_DECLARATION := '0' *)
(* measure the last cycle time and make sure we onle execute once every millisecond *)
tx := T_PLC_MS();
IF NOT init THEN
	init := TRUE;
	last := tx;
	mr.RX := mx;
	mr.R1 := 0.0;
ELSIF tx = last THEN
	RETURN;
ELSE
	tc := DWORD_TO_REAL(tx - last) * 0.001;
END_IF;
last := tx;

(* reset *)
IF rst THEN
	mr.R1 := 0.0;
	mr.RX := 0.0;
ELSE
	(* current consumption measurement *)
	IF I1 THEN MX1 := M1; ELSE MX1 := 0.0; END_IF;
	IF I2 THEN MX2 := M2; ELSE MX2 := 0.0; END_IF;
	(* add up the current values in a double real *)
	MR := R2_ADD(MR,(SEL(I1,0.0,mx1) + SEL(I2, 0.0, mx2)) / D * TC);
	(* set the current output value *)
	MX := mr.RX;
END_IF;

(* revision history

hm	16. sep.2007		rev 1.0
	original version

hm	7. feb 2008		rev 1.1
	use new version of ft_int to avoid a counting stop at high values
	deleted unnecessary limits

hm	24. mar. 2008	rev 1.2
	use data_type real2 to extend accuracy to 15 digits total
	do not use ft_int which adds unnecessary overhead

hm	8. feb. 2009	rev 1.3
	changed mx to be I/O
	make sure calculation works for cycle times < 1 ms

hm	8. mar. 2009	rev 1.4
	last was not updated
	code improvements

*)

END_FUNCTION_BLOCK

(* @NESTEDCOMMENTS := 'Yes' *)
(* @PATH := '\/Engineering\/measurements' *)
(* @OBJECTFLAGS := '0, 8' *)
(* @SYMFILEFLAGS := '2048' *)
FUNCTION_BLOCK METER_STAT
VAR_INPUT
	IN : REAL;
	DI : DATE;
	RST : BOOL;
END_VAR
VAR_IN_OUT
	Last_Day : REAL;
	Current_Day : REAL;
	Last_Week : REAL;
	Current_Week : REAL;
	Last_Month : REAL;
	Current_Month : REAL;
	Last_Year : REAL;
	Current_Year : REAL;
END_VAR
VAR RETAIN
	Year_Start : REAL;
	Month_Start : REAL;
	Week_Start : REAL;
	Day_Start : REAL;
	last_run: DATE;
END_VAR

(*
	version 1.3	18. jul. 2009
	programmer 	oscat
	tested BY		oscat

METER_STAT runs statistics of a metered value, it calculates the current week, day, month and year consumption and stores the corresponding last day, week, month and year value.

*)
(* @END_DECLARATION := '0' *)
IF rst THEN
	Last_Day := 0.0;
	Current_Day := 0.0;
	Day_start := IN;
	Last_week := 0.0;
	Current_week := 0.0;
	Week_start := in;
	Last_month := 0.0;
	Current_month := 0.0;
	month_start := in;
	last_year := 0.0;
	current_year := 0.0;
	year_start := in;
ELSE
	Current_Day := IN - Day_Start;
	Current_Week := In - Week_Start;
	Current_Month := IN - Month_Start;
	Current_Year := IN - Year_Start;
END_IF;

IF YEAR_OF_DATE(DI) > YEAR_OF_DATE(last_run) THEN
	(* a new year has started *)
	last_year := current_year;
	current_year := 0.0;
	year_start := in;
	last_month := current_month;
	current_month := 0.0;
	month_start := in;
	last_day := current_day;
	current_day := 0.0;
	day_start := in;
ELSIF MONTH_OF_DATE(DI) > MONTH_OF_DATE(last_run) THEN
	(* a new month has started, january is alrerady done by year change *)
	last_month := current_month;
	current_month := 0.0;
	month_start := in;
	last_day := current_day;
	current_day := 0.0;
	day_start := in;
ELSIF DAY_OF_YEAR(di) > DAY_OF_YEAR(last_run) THEN
	(* day has chaged, first day of year and first day of month has already been taken care of *)
	last_day := current_day;
	current_day := 0.0;
	day_start := in;
END_IF;
IF DAY_OF_WEEK(DI) < DAY_OF_WEEK(last_run) THEN
	(* a new week has started *)
	last_week := current_week;
	current_week := 0.0;
	week_start := in;
END_IF;
last_run := di;

(* revision history
hm	16. sep. 2007	rev 1.0
	original version

hm	7. oct. 2008	rev 1.1
	changed function year_to_year_of_date
	changed function month to month_of_date
	changed function weekday to day_of_week

hm	11. mar. 2009	rev 1.2
	changed real constants to use dot syntax

hm	18. jul. 2009	rev 1.3
	changes all outputs to be I/O
*)

END_FUNCTION_BLOCK

(* @NESTEDCOMMENTS := 'Yes' *)
(* @PATH := '\/Engineering\/measurements' *)
(* @OBJECTFLAGS := '0, 8' *)
(* @SYMFILEFLAGS := '2048' *)
FUNCTION_BLOCK ONTIME
VAR_INPUT
	IN : BOOL;
	RST : BOOL;
END_VAR
VAR_IN_OUT
	SECONDS : UDINT;
	CYCLES : UDINT;
END_VAR
VAR
	tx: DWORD;
	last : DWORD;
	edge : BOOL;
	init: BOOL;
	ms: DWORD;
END_VAR

(*
version 2.5	18. mar. 2011
programmer 	oscat
tested by		tobias

ONTIME measures the ontime of a signal in seconds.
the output SECONDS is of type DWORD which results in a total measurement range of 1 second up to 136 years.
internally ontime works with a resolution of milliseconds

*)
(* @END_DECLARATION := '0' *)
(* read system time *)
tx := T_PLC_MS();

(* make sure the first cycle works correctly *)
IF NOT init THEN
	init := TRUE;
	last := tx;
	ms := 0;
END_IF;
IF RST THEN
	SECONDS := 0;
	CYCLES := 0;
	last := tx;
	ms := 0;
ELSIF IN THEN
	(* add the current milliseconds *)
	ms := (tx - last) + ms;
	IF ms >= 1000 THEN
		seconds := seconds + 1;
		ms := ms - 1000;
	END_IF;
	cycles := cycles + BOOL_TO_UINT(NOT edge);
END_IF;
last := tx;
edge := in;

(* revision history
hm 22.2.2007		rev 1.1
	changed VAR RETAIN PERSISTENT to VAR RETAIN for better compatibility
	wago lon contollers do not support persisitent

hm 2.8.2007		rev 1.2
	adding time up in a real number will automatically lead to the point where
	small time scales like the cycle time will be below the resolution of real and therefore
	ontime would not increase in small steps as necessary
	the time is now measured internally in two  dwords and be converted to real only for
	output purposes.
	deleted the variable power because it was unnecessary

hm	16.9.2007		rev 1.3
	changes time() to T_plc_ms() for compatibility reasons

hm	2. dec. 2007	rev 1.4
	chaged code for better performance

hm	16. mar. 2008	rev 1.5
	added type conversions to avoid warnings under codesys 3.0

hm	21. oct. 2008	rev 2.0
	changed module for much better performance and allow for external result storage

hm	10. nov. 2008	rev 2.1
	increased internal resolution to milliseconds

hm	16. nov. 2008	rev 2.2
	changed typecast to avoid warnings

hm	17. dec. 2008	rev 2.3
	fixed an error when in would be true for more then 49 days

hm	17. jan 2011	rev 2.4
	init will not clear seconds and cycles, only rst clears these values

hm	18. mar. 2011	rev 2.5
	reset was not working

*)
END_FUNCTION_BLOCK

(* @NESTEDCOMMENTS := 'Yes' *)
(* @PATH := '\/Engineering\/measurements' *)
(* @OBJECTFLAGS := '0, 8' *)
(* @SYMFILEFLAGS := '2048' *)
FUNCTION T_PLC_MS : DWORD
VAR CONSTANT
	debug : BOOL := 0;
	N : INT := 0;
	offset : DWORD := 0;
END_VAR
VAR
	tx : TIME;
END_VAR

(*
version 1.2	16. nov 2008
programmer 	hugo
tested by	oscat

T_PLC_MS reads the internal PLC timer and return the time, it has the advantage to be able to set a debug mode
and speed up the counter to test the plc timer overrun which occurs every 50 days respectively 25 days at siemens S7
this routine also allows to correct the behavior of s7 where the internal plc counter will not count all 32 bits.

*)
(* @END_DECLARATION := '0' *)
tx := TIME();
T_PLC_MS := TIME_TO_DWORD(Tx);
(* hier muss die korrektur f�r step7 stattfinden
plctime muss den vollen wertebereich von time ausnutzen:
wenn bei step7 time -24tage bis plus 24 tage ist dann muss der timer auch beim �berlauf auf -24tage springen
und auf keinen fall auf 0 !!!!
f�r siemens muss ein weiterer fb im main eingebunden werden der sicherstellt das alle 32 bits durchgez�hlt werden.
es kann nur ein fb sein den er muss sich das oberste (32te) bit merken.
oder etwa spring s7 bei �berlauf auf -24 tage????? dann w�re keine korrektur n�tig.
*)
IF debug THEN
	T_PLC_MS := (SHL(T_PLC_MS,N) OR SHL(DWORD#1,N)-1) + OFFSET;
END_IF;

(* revision history
hm	14.9.2007	rev 1.0
	original version

hm	12. nov 2007	rev 1.1
	added temporaray variable tx because some compilers could not handle time() as an argument

hm	16. nov. 2008	rev 1.2
	initialized constants with 0 for compatibility reasons
*)
END_FUNCTION

(* @NESTEDCOMMENTS := 'Yes' *)
(* @PATH := '\/Engineering\/measurements' *)
(* @OBJECTFLAGS := '0, 8' *)
(* @SYMFILEFLAGS := '2048' *)
FUNCTION T_PLC_US : DWORD
VAR CONSTANT
	debug : BOOL := 0;
	N : INT := 0;
	offset : DWORD := 0;
END_VAR
VAR
	tx : TIME;
END_VAR

(*
version 1.2	16 nov 2008
programmer 	hugo
tested by	tobias

T_PLC_US reads the internal PLC timer and return the time, it has the advantage to be able to set a debug mode
and speed up the counter to test the plc timer overrun which occurs every 50 days respectively 25 days at siemens S7
this routine also allows to correct the behavior of s7 where the internal plc counter will not count all 32 bits.

*)
(* @END_DECLARATION := '0' *)
tx := TIME();
T_PLC_US := TIME_TO_DWORD(Tx)*1000;
(* hier muss die korrektur f�r step7 stattfinden
plctime muss den vollen wertebereich von time ausnutzen:
wenn bei step7 time -24tage bis plus 24 tage ist dann muss der timer auch beim �berlauf auf -24tage springen
und auf keinen fall auf 0 !!!!
f�r siemens muss ein weiterer fb im main eingebunden werden der sicherstellt das alle 32 bits durchgez�hlt werden.
es kann nur ein fb sein den er muss sich das oberste (32te) bit merken.
oder etwa spring s7 bei �berlauf auf -24 tage????? dann w�re keine korrektur n�tig.
*)
IF debug THEN
	T_PLC_US := (SHL(T_PLC_US,N) OR SHL(DWORD#1,N)-1) + OFFSET;
END_IF;

(* revision history
hm	14.9.2007	rev 1.0
	original version

hm	12. nov 2007	rev 1.1
	added temporaray variable tx because some compilers could not handle time() as an argument

hm	16. nov. 2008	rev 1.2
	initialized constants with 0 for compatibility reasons

*)
END_FUNCTION

(* @NESTEDCOMMENTS := 'Yes' *)
(* @PATH := '\/Engineering\/measurements' *)
(* @OBJECTFLAGS := '0, 8' *)
(* @SYMFILEFLAGS := '2048' *)
FUNCTION_BLOCK TC_MS

VAR_OUTPUT
	TC : DWORD;
END_VAR
VAR
	init: BOOL;
	tx: DWORD;
	last: DWORD;
END_VAR

(*
	version 1.0	13 mar 2008
	programmer 	hugo
	tested by		tobias

TC_MS delivers the time it was last called on the output TC in Milliseconds.

*)
(* @END_DECLARATION := '0' *)
(* read system timer *)
tx := T_PLC_MS();

IF NOT init THEN
	init := TRUE;
	TC := 0;
ELSE
	tc := tx - last;
END_IF;
last := tx;

(* revision history
hm		13. mar. 2008	rev 1.0
	original version

*)

END_FUNCTION_BLOCK

(* @NESTEDCOMMENTS := 'Yes' *)
(* @PATH := '\/Engineering\/measurements' *)
(* @OBJECTFLAGS := '0, 8' *)
(* @SYMFILEFLAGS := '2048' *)
FUNCTION_BLOCK TC_S

VAR_OUTPUT
	TC : REAL;
END_VAR
VAR
	init: BOOL;
	tx: DWORD;
	last: DWORD;
END_VAR

(*
	version 1.2	11. mar. 2009
	programmer 	hugo
	tested by		tobias

TC_S delivers the time it was last called on the output TC in seconds.

*)
(* @END_DECLARATION := '0' *)
(* read system timer *)
tx := T_PLC_US();

IF NOT init THEN
	init := TRUE;
	TC := 0.0;
ELSE
	tc := DWORD_TO_REAL(tx - last)*1.0E-6;
END_IF;
last := tx;

(* revision history
hm	13. mar. 2008	rev 1.0
	original version

hm	16. mar 2008	rev 1.1
	added type conversion to avoid warnings under codesys 3.0

hm	11. mar. 2009	rev 1.2
	changed real constants to use dot syntax

*)

END_FUNCTION_BLOCK

(* @NESTEDCOMMENTS := 'Yes' *)
(* @PATH := '\/Engineering\/measurements' *)
(* @OBJECTFLAGS := '0, 8' *)
(* @SYMFILEFLAGS := '2048' *)
FUNCTION_BLOCK TC_US

VAR_OUTPUT
	TC : DWORD;
END_VAR
VAR
	init: BOOL;
	tx: DWORD;
	last: DWORD;
END_VAR

(*
	version 1.0	13 mar 2008
	programmer 	hugo
	tested by		tobias

TC_US delivers the time it was last called on the output TC in Microseconds.

*)
(* @END_DECLARATION := '0' *)
(* read system timer *)
tx := T_PLC_US();

IF NOT init THEN
	init := TRUE;
	TC := 0;
ELSE
	tc := tx - last;
END_IF;
last := tx;

(* revision history
hm		13. mar. 2008	rev 1.0
	original version

*)

END_FUNCTION_BLOCK

(* @NESTEDCOMMENTS := 'Yes' *)
(* @PATH := '\/Engineering\/sensor' *)
(* @OBJECTFLAGS := '0, 8' *)
(* @SYMFILEFLAGS := '2048' *)
FUNCTION MULTI_IN : REAL
VAR_INPUT
	in_1 : REAL;
	in_2 : REAL;
	in_3 : REAL;
	default : REAL;
	in_min : REAL;
	in_max : REAL;
	mode : BYTE;
END_VAR
VAR
	count: INT;
	F1: BOOL;
	F2: BOOL;
	F3: BOOL;
END_VAR

(*

version 1.4	18. jul. 2009
programmer 	oscat
tested by		oscat

multi_in is a signal conditioning function which can be configured in 8 different ways.
it is used to read multiple sensors for the same value and protect the user from broken sensors or invalid data from sensors.

multi_in can be configured in different ways:
	mode = 0 means the the avg of the 3 inputs is used, this mode is the default mode.
	mode = 1 means in_1 is used.
	mode = 2 means in_2 is used.
	mode = 3 means in_3 is used.
	mode = 4 means default is used.
	mode = 5 means the lowest of the 3 external temperatures is used.
	mode = 6 means the higest externnal temperature is used.
	mode = 7 means the midlle input is used, if there are only two working, the lowest input is used.
	mode > 7 ,eans output is 0 at all times.
	in any config mode, an input higher then in_max or lower then in_min is ignored to prevent values from broken sensors or wires.
	if all inputs are higher then in_max or lower then in_min, a default value (default) is used.
*)

(* @END_DECLARATION := '0' *)
F1 :=  in_1 > in_min AND in_1 < in_max;
F2 :=  in_2 > in_min AND in_2 < in_max;
F3 :=  in_3 > in_min AND in_3 < in_max;

CASE mode OF
0:	count := 0;
	IF F1 THEN
		count := count + 1;
		MULTI_IN := in_1;
	ELSE
		MULTI_IN := 0.0;
	END_IF;
	IF F2 THEN
		count := count + 1;
		MULTI_IN := MULTI_IN + in_2;
	END_IF;
	IF F3 THEN
		count := count + 1;
		MULTI_IN := MULTI_IN + in_3;
	END_IF;
	MULTI_IN := SEL(count = 0, MULTI_IN / INT_TO_REAL(count), default);

1:	MULTI_IN := SEL(F1, default, IN_1);

2:	MULTI_IN := SEL(F2, default, IN_2);

3:	MULTI_IN := SEL(F3, default, IN_3);

4:	MULTI_IN := default;

5:	MULTI_IN := SEL(F1, in_max, IN_1);
	IF F2 AND in_2 < MULTI_IN THEN MULTI_IN := in_2; END_IF;
	IF F3 AND in_3 < MULTI_IN THEN MULTI_IN := in_3; END_IF;
	IF MULTI_IN = in_max THEN MULTI_IN := default; END_IF;

6:	MULTI_IN := SEL(F1, in_min, IN_1);
	IF F2 AND in_2 > MULTI_IN THEN MULTI_IN := in_2; END_IF;
	IF F3 AND in_3 > MULTI_IN THEN MULTI_IN := in_3; END_IF;
	IF MULTI_IN = in_min THEN MULTI_IN := default; END_IF;

7:	IF F1 AND F2 AND F3 THEN MULTI_IN := MID3(in_1, in_2, in_3);
	ELSIF F1 AND F2 THEN MULTI_IN := MIN(in_1, in_2);
	ELSIF F1 AND F3 THEN MULTI_IN := MIN(in_1, in_3);
	ELSIF F2 AND F3 THEN MULTI_IN := MIN(in_2, in_3);
	ELSIF F1 THEN MULTI_IN := in_1;
	ELSIF F2 THEN MULTI_IN := in_2;
	ELSIF F3 THEN MULTI_IN := in_3;
	ELSE MULTI_IN := default;
	END_IF;

END_CASE;

(*
hm 1.1.2007		rev 1.1
	changed midr to mid3 function

hm	14. 10. 2008	rev 1.2
	corrected an error for in_3 overrange detection
	improved performance

hm	11. mar. 2009	rev 1.3
	changed real constants to use dot syntax

hm	18. jul. 2009	rev 1.4
	improved performance
*)
END_FUNCTION

(* @NESTEDCOMMENTS := 'Yes' *)
(* @PATH := '\/Engineering\/sensor' *)
(* @OBJECTFLAGS := '0, 8' *)
(* @SYMFILEFLAGS := '2048' *)
FUNCTION RES_NI : REAL
VAR_INPUT
	T : REAL;
	R0 : REAL;
END_VAR
VAR CONSTANT
	A : REAL := 0.5485;
	B : REAL := 0.665E-3;
	C : REAL := 2.805E-9;
END_VAR
VAR
	T2: REAL;
END_VAR

(*
version 1.2	2 dec 2007
programmer 	hugo
tested by		tobias

this function returs the resistance for a nickel sensor for a temperature range from -60..+180 �C *)
(* @END_DECLARATION := '0' *)
T2 := T * T;
RES_NI := R0 + A * T + B * T2 + C * T2 * T2;

(* revision history

hm	4.8.2006		rev 1.0
	original version

hm	13.9.2007		rev 1.1
	changed coding for better performance

hm	2. dec. 2007	rev 1.2
	changed code for better performance
*)

(*

 Auszug aus DIN 43760 f�r Ni100

�C		R		�C		R		�C	R		�C		R		�C		R

-60 	69,5 	-10 	94,6 	40 	123,0 	90 		154,9 	140 	190,9
-55 	71,9 	-5 		97,3 	45 	126,0 	95 		158,3 	145 	194,8
-50 	74,3 	0 		100,0 	50 	129,1 	100 	161,8 	150 	198,7
-45 	76,7 	5 		102,8 	55 	132,2 	105 	165,3 	155 	202,6
-40 	79,1 	10 		105,6 	60 	135,3 	110 	168,8 	160 	206,6
-35 	81,6 	15 		108,4 	65 	138,5 	115 	172,4 	165 	210,7
-30 	84,2 	20 		111,2 	70 	141,7 	120 	176,0 	170 	214,8
-25 	86,7 	25 		114,1 	75 	145,0 	125 	179,6 	175 	219,0
-20 	89,3 	30 		117,1 	80 	148,3 	130 	183,3 	180 	223,2
-15 	91,9 	35 		120,0 	85 	151,6 	135 	187,1

*)
END_FUNCTION

(* @NESTEDCOMMENTS := 'Yes' *)
(* @PATH := '\/Engineering\/sensor' *)
(* @OBJECTFLAGS := '0, 8' *)
(* @SYMFILEFLAGS := '2048' *)
FUNCTION RES_NTC : REAL
VAR_INPUT
	T : REAL;
	RN : REAL;
	B : REAL;
END_VAR

(*
version 1.1	11. mar. 2009
programmer 	hugo
tested by		tobias

this function returs the resistance for a NTC sensor for a given temperature in �C.
RN is the resistance at 25 �C and B is a constant for the given sensor.

*)
(* @END_DECLARATION := '0' *)
RES_NTC := RN * EXP(B * (1.0 / (T+273.15) - 0.00335401643468053));

(* revision history

hm 30. dec. 2008	rev 1.0
	original version

hm	11. mar. 2009	rev 1.1
	changed real constants to use dot syntax

*)
END_FUNCTION

(* @NESTEDCOMMENTS := 'Yes' *)
(* @PATH := '\/Engineering\/sensor' *)
(* @OBJECTFLAGS := '0, 8' *)
(* @SYMFILEFLAGS := '2048' *)
FUNCTION RES_PT : REAL
VAR_INPUT
	T : REAL;
	R0 : REAL;
END_VAR
VAR CONSTANT
	A : REAL := 3.90802E-3 ;
	B : REAL := -5.802E-7;
	C : REAL := -4.27350E-12;
END_VAR
VAR
	T2: REAL;
END_VAR

(*
version 1.3	11. mar. 2009
programmer 	hugo
tested by		oscat

this function returs the resistance for a platinum sensor for a temperature range from -200..+850 �C *)
(* @END_DECLARATION := '0' *)
T2 := T * T;

IF T >= 0.0 THEN
	RES_PT := R0 * ( 1.0 + A * T + B * T2);
ELSE
	RES_PT := R0 * ( 1.0 + A * T + B * T2 + C * (T - 100.0) * T2 * T);
END_IF;

(* revision history
hm	4. aug. 2006	rev 1.1
	original version

hm	2. dec 2007	rev 1.2
	changed code for better performance

hm	11. mar. 2009	rev 1.3
	changed real constants to use dot syntax

*)

(*
 Auszug aus DIN 43760 f�r Pt100

�C		R		�C		R		�C	R			�C		R			�C		R			�C		R

-200 	18,49 	-100 	60,25 	0 	100,00 	100 	138,50 	200 	175,84 	300 	212,02
-195 	20,65 	-95 	62,28 	5 	101,95 	105 	140,39 	205 	177,68 	305 	213,80
-190 	22,80 	-90 	64,30 	10 	103,90 	110 	142,29 	210 	179,51 	310 	215,57
-185 	24,94 	-85 	66,31 	15 	105,85 	115 	144,17 	215 	181,34 	315 	217,35
-180 	27,08 	-80 	68,33 	20 	107,79 	120 	146,06 	220 	183,17 	320 	219,12
-175 	29,20 	-75 	70,33 	25 	109,73 	125 	147,94 	225 	184,99 	325 	220,88
-170 	31,32 	-70 	72,33 	30 	111,67 	130 	149,82 	230 	186,82 	330 	222,65
-165 	33,43 	-65 	74,33 	35 	113,61 	135 	151,70 	235 	188,63 	335 	224,41
-160 	35,33 	-60 	76,33 	40 	115,54 	140 	153,58 	240 	190,45 	340 	226,17
-155 	37,63 	-55 	78,32 	45 	117,47 	145 	155,45 	245 	192,26 	345 	227,92
-150 	39,71 	-50 	80,31 	50 	119,40 	150 	157,31 	250 	194,07 	350 	229,67
-145 	41,79 	-45 	82,29 	55 	121,32 	155 	159,18 	255 	195,88 	355 	231,42
-140 	43,87 	-40 	84,27 	60 	123,24 	160 	161,04 	260 	197,69 	360 	233,17
-135 	45,94 	-35 	86,25 	65 	125,16 	165 	162,90 	265 	199,49 	365 	234,91
-130 	48,00 	-30 	88,22 	70 	127,07 	170 	164,76 	270 	201,29 	370 	236,65
-125 	50,06 	-25 	90,19 	75 	128,98 	175 	166,61 	275 	203,08 	375 	238,39
-120 	52,11 	-20 	92,16 	80 	130,89 	180 	168,46 	280 	204,88 	380 	240,13
-115 	54,15 	-15 	94,12 	85 	132,80 	185 	170,31 	285 	206,67 	385 	241,86
-110 	56,19 	-10 	96,09 	90 	134,70 	190 	172,16 	290 	208,45 	390 	243,59
-105 	58,22 	-5 		98,04 	95 	136,60 	195 	174,00 	295 	210,24 	395 	245,31

*)
(*
revision history

*)
END_FUNCTION

(* @NESTEDCOMMENTS := 'Yes' *)
(* @PATH := '\/Engineering\/sensor' *)
(* @OBJECTFLAGS := '0, 8' *)
(* @SYMFILEFLAGS := '2048' *)
FUNCTION RES_SI : REAL
VAR_INPUT
	T : REAL;
	RS : REAL;
	TS : REAL;
END_VAR
VAR CONSTANT
	A : REAL := 7.64E-3;
	B : REAL := 1.66E-5;
END_VAR
VAR
	TX: REAL;
END_VAR

(*
version 1.2	11. mar. 2009
programmer 	hugo
tested by		tobias

this function returs the resistance for a silicon sensor for a temperature range from -50..+150 �C
for example KTY10 normaly Rs at 25 �C
*)
(* @END_DECLARATION := '0' *)
TX := T - TS;
RES_SI := RS * ( 1.0 + A * TX + B * TX * TX);

(* revision history
hm	4. aug 2006	rev 1.0
	original version

hm	2. dec 2007	rev 1.1
	changed code for better performance

hm	11. mar. 2009	rev 1.2
	changed real constants to use dot syntax

*)
END_FUNCTION

(* @NESTEDCOMMENTS := 'Yes' *)
(* @PATH := '\/Engineering\/sensor' *)
(* @OBJECTFLAGS := '0, 8' *)
(* @SYMFILEFLAGS := '2048' *)
FUNCTION SENSOR_INT : REAL
VAR_INPUT
	Voltage : REAL;
	Current : REAL;
	RP : REAL;
	RS : REAL;
END_VAR
VAR
	RG: REAL;
END_VAR

(*
version 1.3	11. mar. 2009
programmer 	hugo
tested by		tobias

this function calculates the real resistance of a sensor RX given a parasitic resistor in parallel to the sensor and an additional serial resistor.
for example a parasitic parallel resistor for a PT100 can be ignored but a series resistor is the cable to the sensor.
for a humidity sensor, the parallel resistor is more dramatic and needs to be considered.
the function allows to consider a parallel and serial resistor at the same time.
with this function and known parasitic serial and parallel resistors the true resistance of the sensor can be calculated.

*)
(* @END_DECLARATION := '0' *)
IF current <> 0.0 THEN
	RG := voltage / current;
	SENSOR_INT := RP * ( RG - RS) / ( RP + RS - RG);
END_IF;

(* revisaion history

hm 20.1.2007		rev 1.1
	deleted input R0 which was not needed.

hm	2. dec 2007	rev 1.2
	corrected an error in formula and improoved speed

hm	11. mar. 2009	rev 1.3
	changed real constants to use dot syntax

*)
END_FUNCTION

(* @NESTEDCOMMENTS := 'Yes' *)
(* @PATH := '\/Engineering\/sensor' *)
(* @OBJECTFLAGS := '0, 8' *)
(* @SYMFILEFLAGS := '2048' *)
FUNCTION TEMP_NI : REAL
VAR_INPUT
	Res : REAL;
	R0 : REAL;
END_VAR

(*
version 1.5	10. mar. 2009
programmer 	hugo
tested by		tobias

this function returns the temperature for a nickel sensor in a range from -60..+180 �C *)
(* @END_DECLARATION := '0' *)
TEMP_NI := (SQRT(0.30085225 - 2.66E-3 * (R0 - Res)) - 0.5485) * 751.8796992;

(* revision history

hm 24.1.2007		rev 1.1
	deleted unused variable A, B, C

hm 10.9.2007		rev 1.2
	changed accuracy to 0.02 degrees to improove performace

hm 17. 12 2007	rev 1.3
	improovements for better performance and higher accuracy

hm	6. jan 2008	rev 1.4
	further performance improvement

hm	10. mar. 2009	rev 1.5
	removed nested comments

*)

END_FUNCTION

(* @NESTEDCOMMENTS := 'Yes' *)
(* @PATH := '\/Engineering\/sensor' *)
(* @OBJECTFLAGS := '0, 8' *)
(* @SYMFILEFLAGS := '2048' *)
FUNCTION TEMP_NTC : REAL
VAR_INPUT
	RES : REAL;
	RN : REAL;
	B : REAL;
END_VAR

(*
version 1.1	11. mar. 2009
programmer 	hugo
tested by		tobias

this function returs the temperature for a NTC sensor for a range from 0..85 �C.
RN is the resistance at 25 �C and B is a constant for the given sensor.

*)
(* @END_DECLARATION := '0' *)
IF res > 0.0 THEN
	TEMP_NTC := B * 298.15 / (B + LN(RES / RN) * 298.15) -273.15;
END_IF;

(* revision history

hm 30. dec. 2008	rev 1.0
	original version

hm	11. mar. 2009	rev 1.1
	changed real constants to use dot syntax

*)
END_FUNCTION

(* @NESTEDCOMMENTS := 'Yes' *)
(* @PATH := '\/Engineering\/sensor' *)
(* @OBJECTFLAGS := '0, 8' *)
(* @SYMFILEFLAGS := '2048' *)
FUNCTION TEMP_PT : REAL
VAR_INPUT
	Res : REAL;
	R0 : REAL;
END_VAR
VAR CONSTANT
	A : REAL := 3.9083E-3 ;
	B : REAL := -5.775E-7;
	accuracy : REAL := 0.01;
END_VAR
VAR
	step: REAL := 50.0;
	X: REAL;
	Y: REAL;
	t1: REAL;
	pt : REF_TO DWORD;
END_VAR

(*
version 1.7	11. mar. 2009
programmer 	hugo
tested by		oscat

this function returs the temperature for a platinum sensor for a range from -200..+850 �C *)
(* @END_DECLARATION := '0' *)
X := A * R0;
Y := B * R0;
IF Res >= R0 THEN
	t1 := X * X - 4.0 * Y * (R0 - Res);
	IF t1 < 0.0 THEN
		TEMP_PT := 10000.0;
	ELSE
		TEMP_PT := (-X + SQRT(t1)) / (2.0 * Y);
	END_IF;
ELSE
	pt := REF(step);
	(* since the formula cannot be solved this is a successive approximation *)
	TEMP_PT := -100.0;
	WHILE step > accuracy DO
		(* test if result greater or less *)
		IF RES_PT(TEMP_PT, R0) < res THEN TEMP_PT := TEMP_PT + step; ELSE TEMP_PT := TEMP_PT - step; END_IF;
		pt^ := pt^ - 8388608;  (* this is a super fast divide by 2 method for non floating point CPUs *)
		(* the alternative code: step := step * 0.5; *)
	END_WHILE;
END_IF;

(* revision history

rev 1.1 hm 24.1.2007
	deleted unused variable C

rev 1.2 hm 10.9.2007
	reduced accuracy to 0.02 to shorten execution time

rev 1.3	hm	2. dec 2007
	changed code for better performance

rev	1.4	hm	23. dec 2007
	avoid a negative square root if input values are wrong

rev 1.5 hm	5. jan 2008
	replaced / 2 with * 0.5 for better performance

hm	31. oct. 2008	rev 1.6
	improved performance

hm	11. mar. 2009	rev 1.7
	changed real constants to use dot syntax

*)

END_FUNCTION

(* @NESTEDCOMMENTS := 'Yes' *)
(* @PATH := '\/Engineering\/sensor' *)
(* @OBJECTFLAGS := '0, 8' *)
(* @SYMFILEFLAGS := '2048' *)
FUNCTION TEMP_SI : REAL
VAR_INPUT
	Res : REAL;
	RS : REAL;
	TS : REAL;
END_VAR

(*
version 1.5	10. mar. 2009
programmer 	hugo
tested by		tobias

this function returs the temperature for a silicon sensor for a range from -60..+180 �C
for example KTY10 RS at TS normally 25 �C
*)
(* @END_DECLARATION := '0' *)
TEMP_SI := (-7.64E-3 + SQRT(Res / RS * 6.64E-5 - 0.803E-5)) * 30120.48193 + TS;

(* revision history

hm 24.1.2007		rev 1.1
	the function would only work for TS = 25, now it works for other values of ts.

hm 10.9.2007		rev 1.2
	changed the function to use successive approcimation to avoid an error generated by a sqrt from a negative result.
	changed accuracy to 0.02 degrees to shorten execution time

hm 17. 12 2007	rev 1.3
	improovements for better performance

hm	6. jan 2008	rev 1.4
	further performance improvement

hm	10. mar. 2009	rev 1.5
	removed nested comments

*)
END_FUNCTION

(* @NESTEDCOMMENTS := 'Yes' *)
(* @PATH := '\/Engineering\/signal generators' *)
(* @OBJECTFLAGS := '0, 8' *)
(* @SYMFILEFLAGS := '2048' *)
FUNCTION_BLOCK _RMP_B
VAR_INPUT
	DIR : BOOL;  (* true = up *)
	E : BOOL := TRUE;
	TR : TIME;
END_VAR
VAR_IN_OUT
	RMP : BYTE;
END_VAR
VAR
	tx, tl, tn : TIME;
	init : BOOL;
	last_dir : BOOL;
	start : BYTE;
END_VAR

(*
version 1.2		19. feb. 2011
programmer 	hugo
tested by		oscat

_RMP_B generates a ramp on an external var of type byte
tr is the total ramp time, E is an enable and dir the direction of the ramp

*)
(* @END_DECLARATION := '0' *)
(* read system timer *)
tx := DWORD_TO_TIME(T_PLC_MS());

IF E AND init AND (dir = last_dir) AND (RMP <> SEL(DIR, 0, 255)) AND TR = tn THEN
	RMP := FRMP_B(start, DIR, tx - tl, TR);
ELSE
	init := TRUE;
	tl := tx;
	tn := tr;
	start := RMP;
END_IF;
last_dir := dir;

(* revison history
hm	22. oct. 2008	rev 1.0
	original version

hm	20. nov. 2008	rev 1.1
	set default for E to be TRUE
	added init

hm	19. nov. 2011	rev 1.2
	new code
*)
END_FUNCTION_BLOCK

(* @NESTEDCOMMENTS := 'Yes' *)
(* @PATH := '\/Engineering\/signal generators' *)
(* @OBJECTFLAGS := '0, 8' *)
(* @SYMFILEFLAGS := '2048' *)
FUNCTION_BLOCK _RMP_NEXT
VAR_INPUT
	E : BOOL := TRUE;
	IN : BYTE;
	TR : TIME;
	TF : TIME;
	TL : TIME;
END_VAR
VAR_OUTPUT
	DIR : BOOL;    (* upwards = TRUE *)
	UP : BOOL;
	DN : BOOL;
END_VAR
VAR_IN_OUT
	OUT : BYTE;
END_VAR
VAR
	rmx : _RMP_B;
	dirx : TREND_DW;
	t_lock :TP;
	xen: BOOL;
	xdir: BOOL;
END_VAR

(*
version 1.4		18. jul. 2009
programmer 	hugo
tested by		oscat

_RMP_NEXT  will generate a ramp output following the input IN.
on a rising ramp the output will stop as soon as it has surpassed the input in, and on a falling ramp it will stop when out is smaller than in.
a lockout time T_L will be added between up and down direction.

*)
(* @END_DECLARATION := '0' *)
dirx(X := in);

t_lock(in := FALSE, pt := TL);

IF dirx.TU AND (OUT < IN) THEN
	IF NOT xdir AND xen THEN t_lock(in := TRUE); END_IF;
	xen := TRUE;
	xdir := TRUE;
ELSIF dirx.TD AND (OUT > IN) THEN
	IF xdir AND xen THEN t_lock(in := TRUE); END_IF;
	xen := TRUE;
	xdir := FALSE;
ELSIF xen THEN
	IF (xdir AND (out >= in)) OR (NOT xdir AND (out <= in)) THEN
		xen := FALSE;
		IF tl > t#0s THEN t_lock(IN := TRUE); END_IF;
	END_IF;
END_IF;

IF NOT t_lock.Q AND xen THEN
		UP := XDIR;
		DIR := XDIR;
		DN := NOT XDIR;
ELSE
	UP := FALSE;
	DN := FALSE;
END_IF;

rmx(rmp := OUT, E := E AND (UP OR DN) , dir := DIR, tr := SEL(dir, TF, TR));

(* revison history
hm	23. nov. 2008	rev 1.0
	original version

hm	24. jan. 2009	rev 1.1
	deleted unused vars tmp1, tmp2

hm	20. feb. 2009	rev 1.2
	improved algorithm
	added TL

hm	9. mar. 2009	rev 1.3
	input E was ignored
	removed double assignments

hm	18. jul. 2009	rev 1.4
	improved performance

*)
END_FUNCTION_BLOCK

(* @NESTEDCOMMENTS := 'Yes' *)
(* @PATH := '\/Engineering\/signal generators' *)
(* @OBJECTFLAGS := '0, 8' *)
(* @SYMFILEFLAGS := '2048' *)
FUNCTION_BLOCK _RMP_W
VAR_INPUT
	DIR : BOOL;
	E : BOOL := TRUE;
	TR : TIME;
END_VAR
VAR_IN_OUT
	RMP : WORD;
END_VAR
VAR
	tx, tl : DWORD;
	step : DINT;
	init: BOOL;
	last_dir : BOOL;
END_VAR

(*
version 1.1	20. nov. 2008
programmer 	hugo
tested by	oscat

_RMP_B generates a ramp on an external var of type byte
tr is the total ramp time, E is an enable and dir the direction of the ramp

*)
(* @END_DECLARATION := '0' *)
tx := T_PLC_MS();
IF E AND init THEN
	(* we need to set tl = tx when direction changes *)
	IF dir XOR last_dir THEN
	 tl := tx;
	 last_dir := dir;
	END_IF;
	(* check_elapsed time and calculate only if necessary *)
	IF tr > t#0s THEN
		step := DWORD_TO_DINT(SHL(tx-tl, 16) / TIME_TO_DWORD(TR));
	ELSE
		step := 65535;
	END_IF;
	IF step > 0 THEN
		(* perform the step on the ramp *)
		tl := tx;
		(* calculate the step response *)
		IF NOT dir THEN step := - step; END_IF;
		rmp := DINT_TO_WORD(LIMIT(0, WORD_TO_DINT(rmp) + step, 65535));
	END_IF;
ELSE
	tl := tx;
	init := TRUE;
END_IF;

(* revison history
hm	22. oct. 2008	rev 1.0
	original version

hm	20. nov. 2008	rev 1.1
	set default for E to be TRUE
	added init

*)
END_FUNCTION_BLOCK

(* @NESTEDCOMMENTS := 'Yes' *)
(* @PATH := '\/Engineering\/signal generators' *)
(* @OBJECTFLAGS := '0, 8' *)
(* @SYMFILEFLAGS := '2048' *)
FUNCTION_BLOCK GEN_PULSE
VAR_INPUT
	ENQ : BOOL := TRUE;
	PTH : TIME;
	PTL : TIME;
END_VAR
VAR_OUTPUT
	Q : BOOL;
END_VAR
VAR
	tx: TIME;
	tn: TIME;
	init: BOOL;
END_VAR

(*
version 1.5	8. apr. 2011
programmer 	hugo
tested by		oscat

GEN_PULSE uses the internal sps timer to generate a continuous output waveform with programmable high and low time.
the accuracy of gen_pulse is depending on the system timer.
when time is 0 the high and low times are exactly one cycle.
ENQ = TRUE will start and ENQ = FALSE will stop the generator.

*)
(* @END_DECLARATION := '0' *)
IF enq THEN
	tx := DWORD_TO_TIME(T_PLC_MS());
	IF NOT init THEN init := TRUE; tn := tx; END_IF;
	IF tx - tn >= SEL(Q, PTL, PTH) THEN
		tn := tn + SEL(Q, PTL, PTH);
		Q := NOT Q;
	END_IF;
ELSE
	Q := FALSE;
	init := FALSE;
END_IF;

(* revision history
hm	29. jun. 2008	rev 1.0
	original version

hm	23. nov. 2008	rev 1.1
	set default for enq to be true

hm	18. jul. 2009	rev 1.2
	improved performance

hm	13. nov. 2009	rev 1.3
	corrected error

hm	16. feb. 2011	rev 1.4
	corrected an error when timer overflows

hm	8. apr. 2011	rev 1.5
	ptl and pth was exchanged
*)
END_FUNCTION_BLOCK

(* @NESTEDCOMMENTS := 'Yes' *)
(* @PATH := '\/Engineering\/signal generators' *)
(* @OBJECTFLAGS := '0, 8' *)
(* @SYMFILEFLAGS := '2048' *)
FUNCTION_BLOCK GEN_PW2
VAR_INPUT
	ENQ : BOOL;
	TH1 : TIME;
	TL1 : TIME;
	TH2 : TIME;
	TL2 : TIME;
	TS : BOOL;
END_VAR
VAR_OUTPUT
	Q : BOOL;
	TH : TIME;
	TL : TIME;
END_VAR
VAR
	t_high : TIME;
	t_low : TIME;
	tx : TIME;
	start : TIME;
	init : BOOL;
	et : TIME;
END_VAR

(*
version 1.1	14. mar. 2009
programmer 	hugo
tested by		oscat

GEN_PW2 generates a time TH? followed by a time TL?.
the input ts selects between 2 sets of timings for the operation.

*)
(* @END_DECLARATION := '0' *)
(* read system timer *)
tx := DWORD_TO_TIME(T_PLC_MS());

(* startup initialization *)
IF NOT init THEN
	start := tx;
	init := TRUE;
	TH := T#0s;
	TL := T#0s;
END_IF;

(* timing selection *)
IF TS THEN
	t_high := TH2;
	t_low := TL2;
ELSE
	t_high := TH1;
	t_low := TL1;
END_IF;

(* normal operation *)
IF ENQ THEN
	et := tx - start;
	IF NOT Q THEN
		IF et >= t_low THEN
			Q := TRUE;
			start := tx;
			TL := T#0s;
		ELSE
			TL := et;
		END_IF;
	ELSE
		IF et >= t_high THEN
			Q := FALSE;
			start := tx;
			TH := T#0s;
		ELSE
			TH := et;
		END_IF;
	END_IF;
ELSE
	Q := FALSE;
	TH := T#0s;
	TL := T#0s;
	start := tx;
END_IF;

(* revision history
hm	26. sep. 2008	rev 1.0
	original version

hm	14. mar. 2009	rev 1.1
	removed double assignments

*)
END_FUNCTION_BLOCK

(* @NESTEDCOMMENTS := 'Yes' *)
(* @PATH := '\/Engineering\/signal generators' *)
(* @OBJECTFLAGS := '0, 8' *)
(* @SYMFILEFLAGS := '2048' *)
FUNCTION_BLOCK GEN_RDM
VAR_INPUT
	PT : TIME;
	AM : REAL := 1;
	OS : REAL;
END_VAR
VAR_OUTPUT
	Q : BOOL;
	Out : REAL;
END_VAR
VAR
	tx : TIME;
	last : TIME;
	init : BOOL;
END_VAR

(*
	version 1.1	16 sep 2007
	programmer 	oscat
	tested BY		oscat

this signal generator generates a random output. The signal is defined by period time (PT),
amplitude (AM), offset (OS).
The Output waveform will have its max peak at AM/2 + OS and its minimum peak at -AM/2 + OS.
The period time PT defines how often the output signal will jump to a new randow value.
The Output Q will be true for one cycle anytime the output OUT has changed

*)
(* @END_DECLARATION := '0' *)
(* read system time and prepare input data *)
tx := DWORD_TO_TIME(T_PLC_MS()) - last;

(* init section *)
IF NOT init THEN
	init := TRUE;
	last := tx;
	tx := t#0s;
END_IF;

(* add last if one cycle is finished *)
IF tx >= pt THEN
	last := last + pt;
	tx := tx - pt;

	(* generate output signal *)
	out := am * (RDM(0) - 0.5) + os;
	q := TRUE;
ELSE
	q := FALSE;
END_IF;

(* revision history

hm	7.2.2007		rev 1.0
	original version

hm	16.9.2007		rev 1.1
	changes time() to T_plc_ms() for compatibility reasons

*)

END_FUNCTION_BLOCK

(* @NESTEDCOMMENTS := 'Yes' *)
(* @PATH := '\/Engineering\/signal generators' *)
(* @OBJECTFLAGS := '0, 8' *)
(* @SYMFILEFLAGS := '2048' *)
FUNCTION_BLOCK GEN_RDT

VAR_INPUT
	Enable		 : BOOL := TRUE ;
	Min_Time_ms	: TIME := t#1s ; (* min Taktzeit *)
	Max_Time_ms	: TIME := t#1.2s ; (* Max Taktzeit *)
	TP_Q		 : TIME := t#100ms ; (* Zeit Ausgang auf TRUE *)
END_VAR
VAR_OUTPUT
	xQ		 : BOOL ;
END_VAR
VAR
	(* Taktgenerator Simulation *)
	tonRDMTimer	: TON ; (* Zeitbaustein Taktgenerator *)
	tof_xQ		: TOF ; (* Ausschaltverz�gerung Taktgenerator *)
	tRDMTime	: TIME ; (* Sollzeit *)
	rRDMTime	: REAL ; (* Zufalswert Timer *)
END_VAR

(*
version 1.1	16 mar. 2008
programmer 	J. Schohaus
tested by		Hugo

RDMT generates a defined pulse with pulse width TP_Q at random times. the random time will be defined with an minimum and maximum time.

*)

(*
FUNCTION_BLOCK RDMTimer
###############################################################################
		 Ersteller / author :		 		 		 		 		 J.Schohaus
		 Datum / date:		 		 		 		 		 		 13.07.2007
###############################################################################
		 �nderungen / Datum / Ersteller :
		 moditication / date / author :
###############################################################################
		 Verwendete Bibliotheken		 ( * werden im Baustein nicht ben�tigt )
		 		 		 		 Oscat.lib
###############################################################################
Beschreibung:
*)
(* @END_DECLARATION := '0' *)
tonRDMTimer ( IN:= Enable , PT:= tRDMTime );
tof_xQ ( IN:= tonRDMTimer.Q , PT:= TP_Q );
XQ := tof_xq.Q;
IF tonRDMTimer.Q THEN
		 xQ := TRUE ;
		 rRDMTime := RDM ( last:= rRDMTime ) ;
		 tRDMTime := REAL_TO_TIME ( rRDMTime * DINT_TO_REAL(TIME_TO_DINT( Max_Time_ms - Min_Time_ms ) + TIME_TO_DINT(Min_Time_ms ))) ;
		 tonRDMTimer ( IN:= FALSE );
END_IF;

(* revision history
J. Schohaus	19. nov 2007	rev 1.0
	origial version

hm	16. mar. 2008			rev 1.1
	added type conversion to avoid warnings under codesys 3.0
*)
END_FUNCTION_BLOCK

(* @NESTEDCOMMENTS := 'Yes' *)
(* @PATH := '\/Engineering\/signal generators' *)
(* @OBJECTFLAGS := '0, 8' *)
(* @SYMFILEFLAGS := '2048' *)
FUNCTION_BLOCK GEN_RMP
VAR_INPUT
	PT : TIME := t#1s;
	AM : REAL := 1.0;
	OS : REAL;
	DL : REAL;
END_VAR
VAR_OUTPUT
	Q : BOOL;
	OUT : REAL;
END_VAR
VAR
	tx : TIME;
	last : TIME;
	init : BOOL;
	temp : REAL;
	ltemp: REAL;
END_VAR

(*
	version 1.4	10. mar. 2009
	programmer 	oscat
	tested BY		oscat

this signal generator generates a ramp wave output. The ramp wave signal is defined by period time (PT),
amplitude (AM), offset (OS) and a specific delay for the output signal (DL).
The Output waveform will have its minimum peak at OS and its maximum peak at AM + OS.
The delay input can delay a signal up to PT, this can be useful to synchronize different generators
and generate interleaving signals.
in addition to the analog output Out there is a second boolean output Q with is true for one cycle when the ramp starts.
*)
(* @END_DECLARATION := '0' *)
(* read system time and prepare input data *)
tx := DWORD_TO_TIME(T_PLC_MS()) - last;
DL := MODR(dl,1.0);
IF dl < 0.0 THEN dl := 1.0 - dl; END_IF;

(* init section *)
IF NOT init THEN
	init := TRUE;
	last := tx;
	tx := t#0s;
END_IF;

(* add last if one cycle is finished *)
IF tx >= pt THEN
	last := last + pt;
	tx := tx - pt;
END_IF;

(* generate sine wave *)
ltemp := temp;
IF pt > t#0s THEN temp := FRACT(TIME_TO_REAL(tx + MULTIME(pt, dl)) / TIME_TO_REAL(pt)); END_IF;
out := am * temp + os;

(* boolean output Q *)
Q := temp < ltemp;

(* revision history
hm	3. mar 2007		rev 1.0
	original version

hm	17 sep 2007		rev 1.1
	replaced time() with t_plc_ms for compatibilitx reasons

hm	27. nov 2007	rev 1.2
	avoid divide by 0 when pt = 0

ks	26. oct. 2008	rev 1.3
	code optimization

hm	10. mar. 2009	rev 1.4
	changed real constants to use dot syntax
*)
END_FUNCTION_BLOCK

(* @NESTEDCOMMENTS := 'Yes' *)
(* @PATH := '\/Engineering\/signal generators' *)
(* @OBJECTFLAGS := '0, 8' *)
(* @SYMFILEFLAGS := '2048' *)
FUNCTION_BLOCK GEN_SIN
VAR_INPUT
	PT : TIME;
	AM : REAL := 1.0;
	OS : REAL;
	DL : REAL;
END_VAR
VAR_OUTPUT
	Q : BOOL;
	Out : REAL;
END_VAR
VAR
	tx : TIME;
	last : TIME;
	init : BOOL;
	temp : REAL;
END_VAR

(*
version 1.6	11. mar. 2009
programmer 	oscat
tested BY	oscat

this signal generator generates a sine wave output. The sine wave signal is defined by period time (PT),
amplitude (AM), offset (OS) and a specific delay for the output signal (DL).
The Output waveform will have its max peak at AM/2 + OS and its minimum peak at -AM/2 + OS.
The delay input can delay a signal up to PT, this can be useful to synchronize different generators
and generate interleaving signals. A Cos wave can be generated accordingly.
in addition to a analog output Out there is a second boolean output Q with the corresponding binary signal.
*)
(* @END_DECLARATION := '0' *)
(* read system time and prepare input data *)
tx := DWORD_TO_TIME(T_PLC_MS()) - last;
DL := MODR(dl,1.0);
IF dl < 0.0 THEN dl := 1.0 - dl; END_IF;

(* init section *)
IF NOT init THEN
	init := TRUE;
	last := tx;
	tx := t#0s;
END_IF;

(* add last if one cycle is finished *)
IF tx >= pt THEN
	last := last + pt;
	tx := tx - pt;
END_IF;

(* generate sine wave *)
IF pt > t#0s THEN temp := SIN(math.PI2 * DWORD_TO_REAL(TIME_TO_DWORD(tx + MULTIME(pt, dl))) / DWORD_TO_REAL(TIME_TO_DWORD(pt))); END_IF;
out := am * 0.5 *  temp + os;

(* boolean output Q *)
q := NOT SIGN_R(temp);

(* revision history
hm	22. jan 2007	rev 1.0
	original version

hm	17 sep 2007	rev 1.1
	replaced time() with t_plc_ms for compatibilitx reasons

hm	27. nov 2007	rev 1.2
	avoid divide by 0 when pt = 0

hm	6. jan 2008		rev 1.3
	improved performance

hm	16. mar. 2008	rev 1.4
	added type conversion to avoid warnings under codesys 3.0

hm	18. oct. 2008	rev 1.5
	using math constants

hm	11. mar. 2009	rev 1.6
	changed real constants to use dot syntax

*)
END_FUNCTION_BLOCK

(* @NESTEDCOMMENTS := 'Yes' *)
(* @PATH := '\/Engineering\/signal generators' *)
(* @OBJECTFLAGS := '0, 8' *)
(* @SYMFILEFLAGS := '2048' *)
FUNCTION_BLOCK GEN_SQR
VAR_INPUT
	PT : TIME;
	AM : REAL := 1.0;
	OS : REAL;
	DC : REAL := 0.5;
	DL : REAL;
END_VAR
VAR_OUTPUT
	Q : BOOL;
	Out : REAL;
END_VAR
VAR
	tx : TIME;
	last : TIME;
	init: BOOL;
END_VAR

(*
version 1.4	11. mar. 2009
programmer 	oscat
tested BY		oscat

this signal generator generates a square wave output. The square wave signal is defined by period time (PT),
amplitude (AM), offset (OS), duty cycle (DC) and a specific delay for the output signal (DL).
The Output waveform will switch between AM/2 + OS and -AM/2 + OS. The DC input specifies ther duty cycle,
DC = 0 means output is low at all times and 1 means output is high at all times.
The delay input can delay a signal up to PT, this can be useful to synchronize different generators and generate interleaving signals.
in addition to a analog output Out there is a second boolean output Q.
*)
(* @END_DECLARATION := '0' *)
(* check dc = 1 or 0 *)
IF dc = 0.0 THEN
	out := -am * 0.5 + os;
	Q := FALSE;
	RETURN;
ELSIF dc = 1.0 THEN
	out := am * 0.5 + os;
	Q := TRUE;
	RETURN;
END_IF;

(* read system time and prepare input data *)
tx := DWORD_TO_TIME(T_PLC_MS()) - last;
DL := MODR(dl,1.0);
IF dl < 0.0 THEN dl := 1.0 - dl; END_IF;
dc := MODR(dc,1.0);
IF dc < 0.0 THEN dc := 1.0 - dc; END_IF;

(* init section *)
IF NOT init THEN
	init := TRUE;
	last := tx;
	tx := t#0s;
END_IF;

(* add last if one cycle is finished *)
IF tx >= pt THEN
	last := last + pt;
	tx := tx - pt;
END_IF;

(* check if falling or rising edge first *)
IF MULTIME(pt, dl + dc) >= pt THEN
	(* generate falling edge *)
	IF tx >= MULTIME(pt, dl + dc - 1) THEN
		out := -am * 0.5 + os;
		Q := FALSE;
	END_IF;
	(* generate rising edge *)
	IF tx >= MULTIME(pt, dl) THEN
		out := am * 0.5 + os;
		Q := TRUE;
	END_IF;
ELSE
	(* generate rising edge first *)
	IF tx >= MULTIME(pt, dl) THEN
		out := am * 0.5 + os;
		Q := TRUE;
	END_IF;
	(* generate falling edge *)
	IF tx >= MULTIME(pt, dl + dc) THEN
		out := -am * 0.5 +os;
		Q := FALSE;
	END_IF;
END_IF;

(* revision history

hm	12. feb 2007	rev 1.1
	added default value for dc = 0.5

hm	17 sep 2007	rev 1.2
	replaced time() with t_plc_ms for compatibilitx reasons

hm	6. jan 2008	rev 1.3
	improved performance

hm	11. mar. 2009	rev 1.4
	changed real constants to use dot syntax
	set default amplitude to 1.0

*)

END_FUNCTION_BLOCK

(* @NESTEDCOMMENTS := 'Yes' *)
(* @PATH := '\/Engineering\/signal generators' *)
(* @OBJECTFLAGS := '0, 8' *)
(* @SYMFILEFLAGS := '2048' *)
FUNCTION_BLOCK PWM_DC
VAR_INPUT
	F : REAL;
	DC : REAL;
END_VAR
VAR_OUTPUT
	Q : BOOL;
END_VAR
VAR
	clk: CLK_PRG;
	pulse: TP_X;
	tmp: REAL;
END_VAR

(*
version 1.4	11. mar. 2009
programmer 	oscat
tested BY		oscat

this signal generator generates a square wave signal which is specified by the frequency and the duty cycle
*)
(* @END_DECLARATION := '0' *)
IF F > 0.0 THEN
	tmp := 1000.0 / F;
	CLK(PT := REAL_TO_TIME(tmp));
	Pulse(in := clk.Q, pt := REAL_TO_TIME(tmp * DC));
	Q := pulse.Q;
END_IF;

(* revision history

hm	25. feb 2007	rev 1.1
	recoded in st for better performance and better portability

hm	27. nov 2007	rev 1.2
	avoid divide by 0 when F = 0

hm	19. oct. 2008	rev 1.3
	changed type TP_R to TP_X because of name change
	improved performance

hm	11. mar. 2009	rev 1.4
	changed real constants to use dot syntax

*)
END_FUNCTION_BLOCK

(* @NESTEDCOMMENTS := 'Yes' *)
(* @PATH := '\/Engineering\/signal generators' *)
(* @OBJECTFLAGS := '0, 8' *)
(* @SYMFILEFLAGS := '2048' *)
FUNCTION_BLOCK PWM_PW
VAR_INPUT
	F : REAL;
	PW : TIME;
END_VAR
VAR_OUTPUT
	Q : BOOL;
END_VAR
VAR
	clk: CLK_PRG;
	pulse: TP_X;
END_VAR

(*
version 1.5	11. mar. 2009
programmer 	oscat
tested BY		oscat

this signal generator generates a square wave signal which is specified by the frequency and the pulse width.
*)
(* @END_DECLARATION := '0' *)
IF F > 0.0 THEN
	CLK(PT := REAL_TO_TIME(1000.0 / F));
	Pulse(in := clk.Q, pt := pw);
	Q := pulse.Q;
END_IF;

(* revision history

hm	25. feb 2007	rev 1.1
	recoded in st for better performance and better portability

hm	27. nov 2007	rev 1.2
	avoid divide by 0 when F = 0

hm	9. dec 2007		rev 1.3
	corrected an error with F = 0

hm	19. oct. 2008	rev 1.4
	changed type tp_r to TP_x brecause of name change

hm	11. mar. 2009	rev 1.5
	changed real constants to use dot syntax

*)
END_FUNCTION_BLOCK

(* @NESTEDCOMMENTS := 'Yes' *)
(* @PATH := '\/Engineering\/signal generators' *)
(* @OBJECTFLAGS := '0, 8' *)
(* @SYMFILEFLAGS := '2048' *)
FUNCTION_BLOCK RMP_B
VAR_INPUT
	SET0 : BOOL;
	PT : TIME;
	E : BOOL := TRUE;
	UP : BOOL := TRUE;
	RST : BOOL;
END_VAR
VAR_OUTPUT
	OUT : BYTE;
	BUSY: BOOL;
	HIGH : BOOL;
	LOW : BOOL;
END_VAR
VAR
	rmp : _RMP_B;
END_VAR

(*
version 2.0	23. oct. 2008
programmer 	oscat
tested BY	oscat

this ramp generator generates a byte wide ramp with 255 steps
the generator has an asynchronous set and reset
the ramp is controlled by PT which is the total ramp time for a full sweep from 0..255
an UD input controlls the direction Up or Down and the E input enables the ramp generation
a busy output indicates that the ramp is running, busy false means output is stable.
the outputs low and high will be true when the output has reached its max or min value.

*)
(* @END_DECLARATION := '0' *)
(* generate ramp *)
rmp(dir := UP, E := E, TR := PT, rmp := out);

(* set or reset operation *)
IF RST THEN
	out := 0;
ELSIF SET0 THEN
	out := 255;
END_IF;

(* checks for outputs stable and reset or set busy flag *)
low := out = 0;
high := out = 255;
busy := NOT (low OR high) AND E;

(* revision history

hm 5.10.2006	rev 1.1
	added busy output
hm 17.1.2007	rev 1.2
	renamed input ud to up for better usability
	deleted unused variable step

hm	17.9.2007		rev 1.3
	replaced time() with t_plc_ms() for compatibility reasons

hm	28. sep 2007	rev 1.4
	added outputs on and off
	busy is now disabled while en is false
	new coding for higher accuracy and performance

hm	5. oct 2007	rev 1.5
	added statements to allow for PT to be t#0s output jumps to max or min immediately

hm	25. dec 2007	rev 1.6
	improved code for better performance

hm	16. oct. 2008	rev 1.7
	improved code for better performance

hm	18. oct. 2008	rev 1.8
	added type conversion to avoid warnings
	changed input en to e for compatibility reasons

hm	23. oct. 2008	REV 	2.0
	new code using _RMP_B

*)
END_FUNCTION_BLOCK

(* @NESTEDCOMMENTS := 'Yes' *)
(* @PATH := '\/Engineering\/signal generators' *)
(* @OBJECTFLAGS := '0, 8' *)
(* @SYMFILEFLAGS := '2048' *)
FUNCTION_BLOCK RMP_SOFT
VAR_INPUT
	IN : BOOL;
	VAL : BYTE;
END_VAR
VAR_INPUT (* CONSTANT *)
	PT_ON: TIME;
	PT_OFF : TIME;
END_VAR
VAR_OUTPUT
	OUT : BYTE;
END_VAR
VAR
	rmp : _RMP_B;
	tmp: BYTE;
END_VAR

(*
version 2.0	26. oct. 2008
programmer 	oscat
tested BY		oscat

this soft on/off ramp generator generates a soft on and soft off ramp while the max on value is set by the input
the time for a full ramp can be set by config variables for up and down ramp.

*)
(* @END_DECLARATION := '0' *)
tmp := SEL(in, 0, val);
IF tmp > out THEN
	(* we need to ramp down *)
	rmp(dir := TRUE, E := TRUE, TR := PT_ON, rmp := out);
	(* make sure out does not surpass tmp *)
	out := MIN(out, tmp);
ELSIF tmp < out THEN
	(* we need to ramp up *)
	rmp(dir := FALSE, E := TRUE, TR := PT_OFF, rmp := out);
	(* make sure out does not surpass tmp *)
	out := MAX(out, tmp);
ELSE
	(* no ramp necessary *)
	rmp(E := FALSE, rmp := out);
END_IF;

(* revision history

hm 22.1.2007	rev 1.1
	deleted unused variables X1 and I, X2 and X3

hm	17.9.2007	rev 1.2
	replaced time() with t_plc_ms() for compatibility reasons

hm	26. oct. 2008	2.0
	new code using _rmp_b
*)

END_FUNCTION_BLOCK

(* @NESTEDCOMMENTS := 'Yes' *)
(* @PATH := '\/Engineering\/signal generators' *)
(* @OBJECTFLAGS := '0, 8' *)
(* @SYMFILEFLAGS := '2048' *)
FUNCTION_BLOCK RMP_W
VAR_INPUT
	SET0 : BOOL;
	PT : TIME;
	E : BOOL := TRUE;
	UP : BOOL := TRUE;
	RST : BOOL;
END_VAR
VAR_OUTPUT
	out : WORD;
	busy : BOOL;
	high : BOOL;
	low : BOOL;
END_VAR
VAR
	rmp : _RMP_W;
END_VAR

(*
version 2.0	23. oct. 2008
programmer 	oscat
tested BY	oscat

this ramp generator generates a Word wide ramp with 65535 steps
the generator has an asynchronous set and reset
the ramp is controlled by PT which is the total ramp time for a full sweep from 0..65535
an UD input controlls the direction Up or Down and the E input enables the ramp generation
a busy output indicates that the ramp is running, busy false means output is stable.
the outputs low and high will be true when the output has reached its max or min value.
*)
(* @END_DECLARATION := '0' *)
(* generate ramp *)
rmp(dir := UP, E := E, TR := PT, rmp := out);

(* set or reset operation *)
IF RST THEN
	out := 0;
ELSIF SET0 THEN
	out := 65535;
END_IF;

(* checks for outputs stable and reset or set busy flag *)
low := out = 0;
high := out = 65535;
busy := NOT (low OR high) AND E;

(* revision history:

hm 4.10.2006		rev 1.1
	added the busy output which signals that the ramp is running.

hm 22.1.2007		rev 1.2
	deleted unused variable step

hm	17.9.2007		rev 1.3
	replaced time() with t_plc_ms() for compatibility reasons

hm	28. sep 2007	rev 1.4
	added outputs on and off
	busy is now disabled while en is false
	new coding for higher accuracy and performance

hm	5. oct 2007	rev 1.5
	added statements to allow for PT to be t#0s output jumps to max or min immediately

hm	2. dec 2007	rev 1.6
	corrected an error in calculation of step response

hm	25. dec 2007	rev 1.7
	corrected an error while step response was too slow for fast rise times

hm	16. oct. 2008	rev 1.8
	improved performance

hm	18. oct. 2008	rev 1.9
	renamed inout EN to E for compatibility reasons

hm	23. oct. 2008	rev 2.0
	new code using _RMP_W
*)

END_FUNCTION_BLOCK

(* @NESTEDCOMMENTS := 'Yes' *)
(* @PATH := '\/Engineering\/signal processing' *)
(* @OBJECTFLAGS := '0, 8' *)
(* @SYMFILEFLAGS := '2048' *)
FUNCTION AIN : REAL
VAR_INPUT
	in : DWORD;
END_VAR
VAR_INPUT (* CONSTANT *)
	Bits : BYTE;
	sign : BYTE := 255;
	low : REAL;
	high : REAL := 10.0;
END_VAR
VAR CONSTANT
	ff : DWORD := 16#FFFFFFFF;
END_VAR
VAR
	temp1 : DWORD;
	temp2 : DWORD;
	sx : BOOL;
END_VAR

(*
version 1.5	16 mar 2008
programmer 	oscat
tested by		tobias

Ain converts signals from A/D converters or other digital sources to an internal real value
the lowest number of bits are extracted from the input word and the sign will be extracted if available separately.
the output signal is then conditioned to range from low to high values for a 0 to max value on the analog inputs:
for example a 15bit input (bits := 12) with sign at bit 15 (0..15) will deliver 0.0 (low value at 0) for an input value of 2#0000_0000_0000
an input value of 2#1111_1111_1111 will deliver 10.0 on the output (high value set to 10).

*)
(* @END_DECLARATION := '0' *)
(* extract the sign bit *)
IF sign < 32 THEN
	temp1 := SHR(in,sign);
	sx := temp1.0;
ELSE
	sx := FALSE;
END_IF;
temp1 := SHR(ff, 32-bits);
temp2 := in AND temp1;
AIN := (high - low) * DWORD_TO_REAL(temp2) / DWORD_TO_REAL(temp1) + low;
IF sx THEN AIN := -AIN; END_IF;

(* revision history
hm 18.8.2006	rev 1.1
	fixed an error with low value negative and high value 0.

hm 19.1.2007	rev 1.2
	fixed an error with sign bit.

hm	13.9.2007	rev 1.3
	changed code to avoid warning under codesys 2.8.1

hm	2. dec 2007	rev 1.4
	changed code for better performance

hm	16. mar 2008	rev 1.5
	added type conversions to avoid warnings under codesys 30
*)
END_FUNCTION

(* @NESTEDCOMMENTS := 'Yes' *)
(* @PATH := '\/Engineering\/signal processing' *)
(* @OBJECTFLAGS := '0, 8' *)
(* @SYMFILEFLAGS := '2048' *)
FUNCTION_BLOCK AIN1
VAR_INPUT
	in : DWORD;
END_VAR
VAR_INPUT (* CONSTANT *)
	sign_bit : INT := 255;
	error_bit : INT := 255;
	error_code_en : BOOL;
	error_code : DWORD;
	overflow_bit : INT := 255;
	overflow_code_en : BOOL;
	overflow_code : DWORD;
	Bit_0 : INT;
	Bit_N : INT := 31;
	out_min : REAL;
	out_max : REAL := 10.0;
	code_min : DWORD;
	code_max : DWORD := 16#FFFFFFFF;
	error_output : REAL;
	overflow_output : REAL := 10.0;
END_VAR
VAR_OUTPUT
	out : REAL;
	sign : BOOL;
	error : BOOL;
	overflow : BOOL;
END_VAR
VAR
	tB: DWORD;
END_VAR

(*
version 1.3	10. mar. 2009
programmer 	oscat
tested by		tobias

Ain1 converts signals from A/D converters or other digital sources to an internal real value.

*)
(* @END_DECLARATION := '0' *)
(* extract error bit *)
error := ((SHR(in,error_bit) AND 16#0000_0001) = 1) OR (error_code_en AND error_code = in);
IF error THEN
	out := error_output;
	RETURN;
END_IF;

(* strip off the data input *)
tb := SHR(SHL(in, 31 - bit_N), 31 - bit_N + Bit_0);

(* extract overflow bit *)
overflow := ((SHR(in,overflow_bit) AND 16#0000_0001) = 1) OR (overflow_code_en AND overflow_code = in) OR (tb < code_min OR tb > code_max);
IF overflow THEN
	out := overflow_output;
	RETURN;
END_IF;

(* extract sign bit *)
sign := (SHR(in,sign_bit) AND 16#0000_0001) = 1;

(* convert in to out *)
out := (DWORD_TO_REAL(tb - code_min) * (out_max - out_min) / DWORD_TO_REAL(code_max - code_min) + out_min);
IF sign THEN out := out * -1.0; END_IF;

(* revision history
hm	23. feb 2008	rev 1.0
	original version

hm	16. mar 2008	rev 1.1
	added type conversions to avoid warnngs under codesys 30

hm	22. apr. 2008	rev 1.2
	corrected error in formula when code_min was set
	corrected error when sign bit was used
	optimized code for better performance

hm	10. mar. 2009	rev 1.3
	real constants updated to new systax using dot

*)
END_FUNCTION_BLOCK

(* @NESTEDCOMMENTS := 'Yes' *)
(* @PATH := '\/Engineering\/signal processing' *)
(* @OBJECTFLAGS := '0, 8' *)
(* @SYMFILEFLAGS := '2048' *)
FUNCTION AOUT : DWORD
VAR_INPUT
	in : REAL;
END_VAR
VAR_INPUT (* CONSTANT *)
	Bits : BYTE;
	sign : BYTE := 255;
	low : REAL;
	high : REAL := 10.0;
END_VAR
VAR CONSTANT
	ff : DWORD := 2#1;
END_VAR
VAR
	in2 : REAL;
	sx : BOOL;
END_VAR

(*
version 1.4	23 feb 2008
programmer 	oscat
tested by		tobias

this module conditions an internal real value for D/A converter.
Aout converts and internal real value to a word for an D/A converter or other output devices.
The input value is converted to a n-bit wide output and a sign bit is set separately as specified.
the outout min value is set for the specified min input value and the max output is set for the max input value.
an input higher or lower then the max or min value will set the respective max or min value or the output.

*)
(* @END_DECLARATION := '0' *)
(* if sign bit is defined *)
IF sign < 32 THEN
	sx := sign_R(in);
	in2 := ABS(in);
ELSE
	in2 := in;
END_IF;

(* begrenze in auf die zul�ssigen werte *)
in2 := LIMIT(low, in2, high);

(* Berechne den Ausgangswert *)
Aout := REAL_TO_DWORD((in2 - low) / (high - low) * DWORD_TO_REAL(SHL(ff,bits) -1));
IF sx THEN Aout := SHL(ff,sign) OR Aout; END_IF;

(*
revision history

hm 18.1.2007		rev 1.1
	renamed Modul to aout.
	changed Output to 32 Bit max.
	corrected error with sign bit.

hm	13.9.2007		rev 1.2
	changed code to avoid warning under codesys 2.8.1

hm	2. dec 2007		rev 1.3
	changed code for better performance

hm	23. feb 2008	rev 1.4
	changed code for better performance
*)
END_FUNCTION

(* @NESTEDCOMMENTS := 'Yes' *)
(* @PATH := '\/Engineering\/signal processing' *)
(* @OBJECTFLAGS := '0, 8' *)
(* @SYMFILEFLAGS := '2048' *)
FUNCTION AOUT1 : DWORD
VAR_INPUT
	in : REAL;
END_VAR
VAR_INPUT (* CONSTANT *)
	Bit_0 : INT;
	Bit_N : INT := 31;
	sign : INT := 255;
	low : REAL;
	high : REAL := 10.0;
END_VAR
VAR CONSTANT
	ff : DWORD := 2#1;
END_VAR
VAR
	sx: BOOL;
	in2 : REAL;
END_VAR

(*
version 1.0	23 feb 2008
programmer 	oscat
tested by		tobias

this module conditions an internal real value for a D/A converter.

*)
(* @END_DECLARATION := '0' *)
(* if sign bit is defined *)
IF sign < 32 THEN
	sx := SIGN_R(in);
	in2 := ABS(in);
ELSE
	in2 := in;
END_IF;

(* begrenze in auf die zul�ssigen werte *)
in2 := LIMIT(low, in2, high);

(* Berechne den Ausgangswert *)
AOUT1 := SHL(REAL_TO_DWORD((in2 - low) / (high - low) * DWORD_TO_REAL(SHL(ff,bit_n - Bit_0 + 1) -1)),Bit_0);
IF sx THEN AOUT1 := SHL(ff,sign) OR AOUT1; END_IF;

(* revision history
hm	23. feb 2008	rev 1.0
	original version

*)
END_FUNCTION

(* @NESTEDCOMMENTS := 'Yes' *)
(* @PATH := '\/Engineering\/signal processing' *)
(* @OBJECTFLAGS := '0, 8' *)
(* @SYMFILEFLAGS := '2048' *)
FUNCTION BYTE_TO_RANGE : REAL
VAR_INPUT
	X : BYTE;
	low : REAL;
	high : REAL;
END_VAR

(*
version 1.0	9. jan 2008
programmer 	hugo
tested by		tobias

Byte_to_Range converts a Byte into a real between low and high.

*)
(* @END_DECLARATION := '0' *)
BYTE_TO_RANGE := (high - low) * X / 255.0 + low;

(* revision history
hm	9. jan 2008		rev 1.0
	original version

*)

END_FUNCTION

(* @NESTEDCOMMENTS := 'Yes' *)
(* @PATH := '\/Engineering\/signal processing' *)
(* @OBJECTFLAGS := '0, 8' *)
(* @SYMFILEFLAGS := '2048' *)
FUNCTION_BLOCK DELAY
VAR_INPUT
	IN : REAL;
	N : INT;
	RST : BOOL;
END_VAR
VAR_OUTPUT
	OUT : REAL;
END_VAR
VAR
	buf : ARRAY[0..31] OF REAL;
	i : INT;
	init: BOOL;
	stop: INT;
END_VAR

(*
version 1.5	23. mar. 2009
programmer 	hugo
tested by		oscat

this function block delays input values by each programm cycle
after N+1 cycles the in value has shifted to the out.
N can be any alue from 0 .. 32
if n = 0 the input will be present on the output without a delay.
f N > 32 then the output will be delayed by 32 cycles.
any high on rst will load the buffer with in.

*)
(* @END_DECLARATION := '0' *)
stop := LIMIT(0,N,32) - 1;
IF rst OR NOT init THEN
	init := TRUE;
	FOR i := 0 TO stop DO buf[i] := in; END_FOR;
	out := in;
	i := 0;
ELSIF stop < 0 THEN
	out := in;
ELSE
	out := buf[i];
	buf[i] := in;
	i := INC1(i, N);
END_IF;

(* revision history
hm 1.10.2006		rev 1.1
	corrected error in buffer management

hm 19.1.2007		rev 1.2
	changed reset to load the value of in instead of 0
